LIN {X 0,Y 369.061,Z 354.137,A -85,B 0,C 180,E1 -12856.791,E2 -12856.791} C_VEL
LIN {X 0,Y 369.066,Z 354.138,A -85,B 0,C 180,E1 -12860.132,E2 -12860.132} C_VEL
LIN {X 0,Y 369.162,Z 354.122,A -85,B 0,C 180,E1 -12863.442,E2 -12863.442} C_VEL
LIN {X 0,Y 369.306,Z 354.106,A -85,B 0,C 180,E1 -12867.819,E2 -12867.819} C_VEL
LIN {X 0,Y 369.304,Z 354.11,A -85,B 0,C 180,E1 -12872.182,E2 -12872.182} C_VEL
LIN {X 0,Y 369.16,Z 354.127,A -85,B 0,C 180,E1 -12876.56,E2 -12876.56} C_VEL
LIN {X 0,Y 369.069,Z 354.154,A -85,B 0,C 180,E1 -12879.207,E2 -12879.207} C_VEL
LIN {X 0,Y 370.205,Z 357.177,A -85,B 0,C 180,E1 -12879.375,E2 -12879.375} C_VEL
LIN {X 0,Y 381.684,Z 380.076,A -85,B 0,C 180,E1 -12880.832,E2 -12880.832} C_VEL
LIN {X 0,Y 385.674,Z 389.818,A -85,B 0,C 180,E1 -12881.355,E2 -12881.355} C_VEL
LIN {X 0,Y 382.326,Z 514.998,A -85,B 0,C 180,E1 -12883.86,E2 -12883.86} C_VEL
LIN {X 0,Y 381.61,Z 530.295,A -85,B 0,C 180,E1 -12884.372,E2 -12884.372} C_VEL
LIN {X 0,Y 380.673,Z 545.172,A -85,B 0,C 180,E1 -12885.085,E2 -12885.085} C_VEL
LIN {X 0,Y 379.475,Z 558.92,A -85,B 0,C 180,E1 -12885.948,E2 -12885.948} C_VEL
LIN {X 0,Y 378.337,Z 564.266,A -85,B 0,C 180,E1 -12886.294,E2 -12886.294} C_VEL
LIN {X 0,Y 374.743,Z 572.831,A -85,B 0,C 180,E1 -12886.834,E2 -12886.834} C_VEL
LIN {X 0,Y 371.121,Z 581.153,A -85,B 0,C 180,E1 -12887.454,E2 -12887.454} C_VEL
LIN {X 0,Y 369.922,Z 585.999,A -85,B 0,C 180,E1 -12887.926,E2 -12887.926} C_VEL
LIN {X 0,Y 368.194,Z 599.192,A -85,B 0,C 180,E1 -12889.514,E2 -12889.514} C_VEL
LIN {X 0,Y 366.673,Z 609.996,A -85,B 0,C 180,E1 -12891.092,E2 -12891.092} C_VEL
LIN {X 0,Y 365.196,Z 620.539,A -85,B 0,C 180,E1 -12892.936,E2 -12892.936} C_VEL
LIN {X 0,Y 363.939,Z 629.47,A -85,B 0,C 180,E1 -12894.821,E2 -12894.821} C_VEL
LIN {X 0,Y 362.732,Z 637.87,A -85,B 0,C 180,E1 -12896.967,E2 -12896.967} C_VEL
LIN {X 0,Y 361.879,Z 644.548,A -85,B 0,C 180,E1 -12899.079,E2 -12899.079} C_VEL
LIN {X 0,Y 361.278,Z 649.748,A -85,B 0,C 180,E1 -12901.135,E2 -12901.135} C_VEL
LIN {X 0,Y 360.891,Z 653.719,A -85,B 0,C 180,E1 -12903.134,E2 -12903.134} C_VEL
LIN {X 0,Y 360.521,Z 656.543,A -85,B 0,C 180,E1 -12905.039,E2 -12905.039} C_VEL
LIN {X 0,Y 360.316,Z 658.689,A -85,B 0,C 180,E1 -12907.205,E2 -12907.205} C_VEL
LIN {X 0,Y 360.265,Z 659.556,A -85,B 0,C 180,E1 -12908.71,E2 -12908.71} C_VEL
LIN {X 0,Y 360.246,Z 659.917,A -85,B 0,C 180,E1 -12910.46,E2 -12910.46} C_VEL
LIN {X 0,Y 360.31,Z 659.558,A -85,B 0,C 180,E1 -12912.165,E2 -12912.165} C_VEL
LIN {X 0,Y 360.551,Z 657.956,A -85,B 0,C 180,E1 -12914.566,E2 -12914.566} C_VEL
LIN {X 0,Y 361.005,Z 654.876,A -85,B 0,C 180,E1 -12917.048,E2 -12917.048} C_VEL
LIN {X 0,Y 361.53,Z 650.776,A -85,B 0,C 180,E1 -12919.302,E2 -12919.302} C_VEL
LIN {X 0,Y 362.352,Z 645.097,A -85,B 0,C 180,E1 -12921.635,E2 -12921.635} C_VEL
LIN {X 0,Y 363.361,Z 638.585,A -85,B 0,C 180,E1 -12923.741,E2 -12923.741} C_VEL
LIN {X 0,Y 364.596,Z 631.247,A -85,B 0,C 180,E1 -12925.679,E2 -12925.679} C_VEL
LIN {X 0,Y 366.096,Z 622.256,A -85,B 0,C 180,E1 -12927.638,E2 -12927.638} C_VEL
LIN {X 0,Y 367.793,Z 612.196,A -85,B 0,C 180,E1 -12929.452,E2 -12929.452} C_VEL
LIN {X 0,Y 369.643,Z 600.703,A -85,B 0,C 180,E1 -12931.17,E2 -12931.17} C_VEL
LIN {X 0,Y 371.322,Z 589.315,A -85,B 0,C 180,E1 -12932.586,E2 -12932.586} C_VEL
LIN {X 0,Y 373.074,Z 576.772,A -85,B 0,C 180,E1 -12933.874,E2 -12933.874} C_VEL
LIN {X 0,Y 374.714,Z 562.889,A -85,B 0,C 180,E1 -12935.038,E2 -12935.038} C_VEL
LIN {X 0,Y 376.037,Z 549.259,A -85,B 0,C 180,E1 -12935.946,E2 -12935.946} C_VEL
LIN {X 0,Y 377.167,Z 534.242,A -85,B 0,C 180,E1 -12936.716,E2 -12936.716} C_VEL
LIN {X 0,Y 378.025,Z 519.128,A -85,B 0,C 180,E1 -12937.262,E2 -12937.262} C_VEL
LIN {X 0,Y 379.027,Z 486.351,A -85,B 0,C 180,E1 -12937.99,E2 -12937.99} C_VEL
LIN {X 0,Y 382.012,Z 393.164,A -85,B 0,C 180,E1 -12939.942,E2 -12939.942} C_VEL
LIN {X 0,Y 374.44,Z 377.297,A -85,B 0,C 180,E1 -12941.119,E2 -12941.119} C_VEL
LIN {X 0,Y 367.639,Z 365.381,A -85,B 0,C 180,E1 -12942.189,E2 -12942.189} C_VEL
LIN {X 0,Y 363.906,Z 359.129,A -85,B 0,C 180,E1 -12942.798,E2 -12942.798} C_VEL
LIN {X 0,Y 362.223,Z 356.441,A -85,B 0,C 180,E1 -12943.08,E2 -12943.08} C_VEL
LIN {X 0,Y 361.891,Z 355.027,A -85,B 0,C 180,E1 -12943.209,E2 -12943.209} C_VEL
LIN {X 0,Y 362.003,Z 355.019,A -85,B 0,C 180,E1 -12946.528,E2 -12946.528} C_VEL
LIN {X 0,Y 362.002,Z 355.019,A -85,B 0,C 180,E1 -12949.937,E2 -12949.937} C_VEL
LIN {X 0,Y 362.122,Z 355.001,A -85,B 0,C 180,E1 -12953.312,E2 -12953.312} C_VEL
LIN {X 0,Y 362.268,Z 354.984,A -85,B 0,C 180,E1 -12957.776,E2 -12957.776} C_VEL
LIN {X 0,Y 362.383,Z 354.969,A -85,B 0,C 180,E1 -12960,E2 -12960} C_VEL
LIN {X 0,Y 362.28,Z 354.98,A -85,B 0,C 180,E1 -12962.223,E2 -12962.223} C_VEL
LIN {X 0,Y 362.126,Z 355.001,A -85,B 0,C 180,E1 -12966.687,E2 -12966.687} C_VEL
LIN {X 0,Y 362.003,Z 355.012,A -85,B 0,C 180,E1 -12970.062,E2 -12970.062} C_VEL
LIN {X 0,Y 362,Z 355.017,A -85,B 0,C 180,E1 -12973.898,E2 -12973.898} C_VEL
LIN {X 0,Y 361.93,Z 355.024,A -85,B 0,C 180,E1 -12976.934,E2 -12976.934} C_VEL
LIN {X 0,Y 361.896,Z 355.03,A -85,B 0,C 180,E1 -12980.46,E2 -12980.46} C_VEL
LIN {X 0,Y 361.897,Z 355.025,A -85,B 0,C 180,E1 -12984.113,E2 -12984.113} C_VEL
LIN {X 0,Y 361.945,Z 355.023,A -85,B 0,C 180,E1 -12986.721,E2 -12986.721} C_VEL
LIN {X 0,Y 361.876,Z 355.03,A -85,B 0,C 180,E1 -12990.327,E2 -12990.327} C_VEL
LIN {X 0,Y 361.856,Z 355.036,A -85,B 0,C 180,E1 -12994.28,E2 -12994.28} C_VEL
LIN {X 0,Y 361.865,Z 355.035,A -85,B 0,C 180,E1 -12997.222,E2 -12997.222} C_VEL
LIN {X 0,Y 361.837,Z 355.04,A -85,B 0,C 180,E1 -13000.755,E2 -13000.755} C_VEL
LIN {X 0,Y 361.822,Z 355.041,A -85,B 0,C 180,E1 -13004.367,E2 -13004.367} C_VEL
LIN {X 0,Y 361.838,Z 355.039,A -85,B 0,C 180,E1 -13007.567,E2 -13007.567} C_VEL
LIN {X 0,Y 361.871,Z 355.094,A -85,B 0,C 180,E1 -13010.388,E2 -13010.388} C_VEL
LIN {X 0,Y 365.331,Z 366.466,A -85,B 0,C 180,E1 -13013.39,E2 -13013.39} C_VEL
LIN {X 0,Y 368.142,Z 376.652,A -85,B 0,C 180,E1 -13015.863,E2 -13015.863} C_VEL
LIN {X 0,Y 370.196,Z 385.294,A -85,B 0,C 180,E1 -13017.818,E2 -13017.818} C_VEL
LIN {X 0,Y 374.385,Z 395.128,A -85,B 0,C 180,E1 -13018.521,E2 -13018.521} C_VEL
LIN {X 0,Y 378.827,Z 419.388,A -85,B 0,C 180,E1 -13019.578,E2 -13019.578} C_VEL
LIN {X 0,Y 381.127,Z 434.485,A -85,B 0,C 180,E1 -13020.167,E2 -13020.167} C_VEL
LIN {X 0,Y 377.305,Z 553.846,A -85,B 0,C 180,E1 -13022.66,E2 -13022.66} C_VEL
LIN {X 0,Y 376.29,Z 569.415,A -85,B 0,C 180,E1 -13023.181,E2 -13023.181} C_VEL
LIN {X 0,Y 374.756,Z 585.071,A -85,B 0,C 180,E1 -13023.925,E2 -13023.925} C_VEL
LIN {X 0,Y 373.122,Z 599.399,A -85,B 0,C 180,E1 -13024.834,E2 -13024.834} C_VEL
LIN {X 0,Y 371.252,Z 613.643,A -85,B 0,C 180,E1 -13025.983,E2 -13025.983} C_VEL
LIN {X 0,Y 369.261,Z 627.13,A -85,B 0,C 180,E1 -13027.33,E2 -13027.33} C_VEL
LIN {X 0,Y 367.379,Z 639.47,A -85,B 0,C 180,E1 -13028.833,E2 -13028.833} C_VEL
LIN {X 0,Y 365.686,Z 650.7,A -85,B 0,C 180,E1 -13030.474,E2 -13030.474} C_VEL
LIN {X 0,Y 364.14,Z 661.138,A -85,B 0,C 180,E1 -13032.303,E2 -13032.303} C_VEL
LIN {X 0,Y 362.777,Z 670.461,A -85,B 0,C 180,E1 -13034.263,E2 -13034.263} C_VEL
LIN {X 0,Y 361.798,Z 678.215,A -85,B 0,C 180,E1 -13036.23,E2 -13036.23} C_VEL
LIN {X 0,Y 361.144,Z 684.684,A -85,B 0,C 180,E1 -13038.209,E2 -13038.209} C_VEL
LIN {X 0,Y 360.631,Z 690.639,A -85,B 0,C 180,E1 -13040.465,E2 -13040.465} C_VEL
LIN {X 0,Y 360.485,Z 694.219,A -85,B 0,C 180,E1 -13042.156,E2 -13042.156} C_VEL
LIN {X 0,Y 360.396,Z 697.799,A -85,B 0,C 180,E1 -13044.404,E2 -13044.404} C_VEL
LIN {X 0,Y 360.38,Z 700.136,A -85,B 0,C 180,E1 -13046.646,E2 -13046.646} C_VEL
LIN {X 0,Y 360.529,Z 701.285,A -85,B 0,C 180,E1 -13048.883,E2 -13048.883} C_VEL
LIN {X 0,Y 360.529,Z 701.244,A -85,B 0,C 180,E1 -13051.116,E2 -13051.116} C_VEL
LIN {X 0,Y 360.387,Z 699.974,A -85,B 0,C 180,E1 -13053.353,E2 -13053.353} C_VEL
LIN {X 0,Y 360.386,Z 697.46,A -85,B 0,C 180,E1 -13055.595,E2 -13055.595} C_VEL
LIN {X 0,Y 360.479,Z 693.683,A -85,B 0,C 180,E1 -13057.843,E2 -13057.843} C_VEL
LIN {X 0,Y 360.693,Z 688.544,A -85,B 0,C 180,E1 -13060.099,E2 -13060.099} C_VEL
LIN {X 0,Y 361.292,Z 681.924,A -85,B 0,C 180,E1 -13062.355,E2 -13062.355} C_VEL
LIN {X 0,Y 362.189,Z 673.631,A -85,B 0,C 180,E1 -13064.61,E2 -13064.61} C_VEL
LIN {X 0,Y 363.223,Z 664.766,A -85,B 0,C 180,E1 -13066.582,E2 -13066.582} C_VEL
LIN {X 0,Y 364.739,Z 654.106,A -85,B 0,C 180,E1 -13068.537,E2 -13068.537} C_VEL
LIN {X 0,Y 366.115,Z 643.14,A -85,B 0,C 180,E1 -13070.214,E2 -13070.214} C_VEL
LIN {X 0,Y 367.699,Z 631.184,A -85,B 0,C 180,E1 -13071.735,E2 -13071.735} C_VEL
LIN {X 0,Y 369.248,Z 619.571,A -85,B 0,C 180,E1 -13072.965,E2 -13072.965} C_VEL
LIN {X 0,Y 371.086,Z 605.528,A -85,B 0,C 180,E1 -13074.176,E2 -13074.176} C_VEL
LIN {X 0,Y 372.586,Z 591.611,A -85,B 0,C 180,E1 -13075.138,E2 -13075.138} C_VEL
LIN {X 0,Y 373.905,Z 577.102,A -85,B 0,C 180,E1 -13075.913,E2 -13075.913} C_VEL
LIN {X 0,Y 374.933,Z 562.841,A -85,B 0,C 180,E1 -13076.472,E2 -13076.472} C_VEL
LIN {X 0,Y 375.62,Z 547.531,A -85,B 0,C 180,E1 -13076.87,E2 -13076.87} C_VEL
LIN {X 0,Y 378.618,Z 434.526,A -85,B 0,C 180,E1 -13079.154,E2 -13079.154} C_VEL
LIN {X 0,Y 373.667,Z 404.594,A -85,B 0,C 180,E1 -13080.216,E2 -13080.216} C_VEL
LIN {X 0,Y 370.766,Z 389.788,A -85,B 0,C 180,E1 -13080.796,E2 -13080.796} C_VEL
LIN {X 0,Y 370.286,Z 388.239,A -85,B 0,C 180,E1 -13080.906,E2 -13080.906} C_VEL
LIN {X 0,Y 367.141,Z 374.609,A -85,B 0,C 180,E1 -13083.719,E2 -13083.719} C_VEL
LIN {X 0,Y 362.919,Z 358.954,A -85,B 0,C 180,E1 -13087.167,E2 -13087.167} C_VEL
LIN {X 0,Y 361.884,Z 355.037,A -85,B 0,C 180,E1 -13088.077,E2 -13088.077} C_VEL
LIN {X 0,Y 361.825,Z 355.042,A -85,B 0,C 180,E1 -13091.33,E2 -13091.33} C_VEL
LIN {X 0,Y 361.832,Z 355.035,A -85,B 0,C 180,E1 -13094.365,E2 -13094.365} C_VEL
LIN {X 0,Y 361.833,Z 355.037,A -85,B 0,C 180,E1 -13097.568,E2 -13097.568} C_VEL
LIN {X 0,Y 361.867,Z 355.035,A -85,B 0,C 180,E1 -13100.973,E2 -13100.973} C_VEL
LIN {X 0,Y 361.871,Z 355.032,A -85,B 0,C 180,E1 -13104.655,E2 -13104.655} C_VEL
LIN {X 0,Y 361.834,Z 355.035,A -85,B 0,C 180,E1 -13108.371,E2 -13108.371} C_VEL
LIN {X 0,Y 361.897,Z 355.032,A -85,B 0,C 180,E1 -13110.955,E2 -13110.955} C_VEL
LIN {X 0,Y 361.951,Z 355.023,A -85,B 0,C 180,E1 -13113.475,E2 -13113.475} C_VEL
LIN {X 0,Y 361.887,Z 355.034,A -85,B 0,C 180,E1 -13117.145,E2 -13117.145} C_VEL
LIN {X 0,Y 361.903,Z 355.029,A -85,B 0,C 180,E1 -13120.724,E2 -13120.724} C_VEL
LIN {X 0,Y 361.93,Z 355.029,A -85,B 0,C 180,E1 -13123.066,E2 -13123.066} C_VEL
LIN {X 0,Y 361.995,Z 355.016,A -85,B 0,C 180,E1 -13126.528,E2 -13126.528} C_VEL
LIN {X 0,Y 362.028,Z 355.01,A -85,B 0,C 180,E1 -13129.938,E2 -13129.938} C_VEL
LIN {X 0,Y 362.158,Z 354.997,A -85,B 0,C 180,E1 -13133.314,E2 -13133.314} C_VEL
LIN {X 0,Y 362.28,Z 354.979,A -85,B 0,C 180,E1 -13137.777,E2 -13137.777} C_VEL
LIN {X 0,Y 362.425,Z 354.961,A -85,B 0,C 180,E1 -13140,E2 -13140} C_VEL
LIN {X 0,Y 362.28,Z 354.98,A -85,B 0,C 180,E1 -13142.224,E2 -13142.224} C_VEL
LIN {X 0,Y 362.17,Z 354.997,A -85,B 0,C 180,E1 -13146.687,E2 -13146.687} C_VEL
LIN {X 0,Y 362.072,Z 355.011,A -85,B 0,C 180,E1 -13148.934,E2 -13148.934} C_VEL
LIN {X 0,Y 361.958,Z 355.021,A -85,B 0,C 180,E1 -13152.333,E2 -13152.333} C_VEL
LIN {X 0,Y 361.96,Z 355.023,A -85,B 0,C 180,E1 -13154.621,E2 -13154.621} C_VEL
LIN {X 0,Y 361.958,Z 355.02,A -85,B 0,C 180,E1 -13158.1,E2 -13158.1} C_VEL
LIN {X 0,Y 361.859,Z 355.032,A -85,B 0,C 180,E1 -13161.655,E2 -13161.655} C_VEL
LIN {X 0,Y 361.924,Z 355.024,A -85,B 0,C 180,E1 -13165.291,E2 -13165.291} C_VEL
LIN {X 0,Y 361.917,Z 355.024,A -85,B 0,C 180,E1 -13167.779,E2 -13167.779} C_VEL
LIN {X 0,Y 361.845,Z 355.034,A -85,B 0,C 180,E1 -13171.286,E2 -13171.286} C_VEL
LIN {X 0,Y 361.853,Z 355.035,A -85,B 0,C 180,E1 -13174.281,E2 -13174.281} C_VEL
LIN {X 0,Y 361.862,Z 355.032,A -85,B 0,C 180,E1 -13177.223,E2 -13177.223} C_VEL
LIN {X 0,Y 361.833,Z 355.04,A -85,B 0,C 180,E1 -13180.756,E2 -13180.756} C_VEL
LIN {X 0,Y 361.816,Z 355.041,A -85,B 0,C 180,E1 -13184.369,E2 -13184.369} C_VEL
LIN {X 0,Y 361.832,Z 355.035,A -85,B 0,C 180,E1 -13187.57,E2 -13187.57} C_VEL
LIN {X 0,Y 361.864,Z 355.033,A -85,B 0,C 180,E1 -13190.975,E2 -13190.975} C_VEL
LIN {X 0,Y 361.875,Z 355.035,A -85,B 0,C 180,E1 -13194.656,E2 -13194.656} C_VEL
LIN {X 0,Y 361.839,Z 355.039,A -85,B 0,C 180,E1 -13198.371,E2 -13198.371} C_VEL
LIN {X 0,Y 361.867,Z 355.032,A -85,B 0,C 180,E1 -13200.953,E2 -13200.953} C_VEL
LIN {X 0,Y 361.897,Z 355.03,A -85,B 0,C 180,E1 -13204.708,E2 -13204.708} C_VEL
LIN {X 0,Y 361.894,Z 355.033,A -85,B 0,C 180,E1 -13208.348,E2 -13208.348} C_VEL
LIN {X 0,Y 361.907,Z 355.029,A -85,B 0,C 180,E1 -13212.093,E2 -13212.093} C_VEL
LIN {X 0,Y 361.983,Z 355.02,A -85,B 0,C 180,E1 -13216.114,E2 -13216.114} C_VEL
LIN {X 0,Y 362.003,Z 355.016,A -85,B 0,C 180,E1 -13219.938,E2 -13219.938} C_VEL
LIN {X 0,Y 362.125,Z 354.998,A -85,B 0,C 180,E1 -13223.313,E2 -13223.313} C_VEL
LIN {X 0,Y 362.268,Z 354.982,A -85,B 0,C 180,E1 -13227.777,E2 -13227.777} C_VEL
LIN {X 0,Y 362.195,Z 354.99,A -85,B 0,C 180,E1 -13231.112,E2 -13231.112} C_VEL
LIN {X 0,Y 362.267,Z 354.987,A -85,B 0,C 180,E1 -13232.224,E2 -13232.224} C_VEL
LIN {X 0,Y 362.125,Z 355.003,A -85,B 0,C 180,E1 -13236.688,E2 -13236.688} C_VEL
LIN {X 0,Y 362.068,Z 355.008,A -85,B 0,C 180,E1 -13238.599,E2 -13238.599} C_VEL
LIN {X 0,Y 363.202,Z 358.066,A -85,B 0,C 180,E1 -13238.792,E2 -13238.792} C_VEL
LIN {X 0,Y 375.716,Z 382.87,A -85,B 0,C 180,E1 -13240.426,E2 -13240.426} C_VEL
LIN {X 0,Y 379.276,Z 391.483,A -85,B 0,C 180,E1 -13240.904,E2 -13240.904} C_VEL
LIN {X 0,Y 375.837,Z 515.861,A -85,B 0,C 180,E1 -13243.443,E2 -13243.443} C_VEL
LIN {X 0,Y 375.108,Z 530.746,A -85,B 0,C 180,E1 -13243.951,E2 -13243.951} C_VEL
LIN {X 0,Y 374.11,Z 545.881,A -85,B 0,C 180,E1 -13244.692,E2 -13244.692} C_VEL
LIN {X 0,Y 372.819,Z 560.212,A -85,B 0,C 180,E1 -13245.612,E2 -13245.612} C_VEL
LIN {X 0,Y 371.331,Z 574.464,A -85,B 0,C 180,E1 -13246.776,E2 -13246.776} C_VEL
LIN {X 0,Y 369.922,Z 585.999,A -85,B 0,C 180,E1 -13247.926,E2 -13247.926} C_VEL
LIN {X 0,Y 368.73,Z 590.809,A -85,B 0,C 180,E1 -13248.424,E2 -13248.424} C_VEL
LIN {X 0,Y 365.027,Z 598.445,A -85,B 0,C 180,E1 -13249.224,E2 -13249.224} C_VEL
LIN {X 0,Y 361.249,Z 605.781,A -85,B 0,C 180,E1 -13250.096,E2 -13250.096} C_VEL
LIN {X 0,Y 359.922,Z 610.01,A -85,B 0,C 180,E1 -13250.717,E2 -13250.717} C_VEL
LIN {X 0,Y 358.5,Z 619.679,A -85,B 0,C 180,E1 -13252.416,E2 -13252.416} C_VEL
LIN {X 0,Y 357.085,Z 629.183,A -85,B 0,C 180,E1 -13254.414,E2 -13254.414} C_VEL
LIN {X 0,Y 355.95,Z 636.912,A -85,B 0,C 180,E1 -13256.376,E2 -13256.376} C_VEL
LIN {X 0,Y 355.098,Z 643.383,A -85,B 0,C 180,E1 -13258.36,E2 -13258.36} C_VEL
LIN {X 0,Y 354.428,Z 648.754,A -85,B 0,C 180,E1 -13260.375,E2 -13260.375} C_VEL
LIN {X 0,Y 353.956,Z 653.014,A -85,B 0,C 180,E1 -13262.419,E2 -13262.419} C_VEL
LIN {X 0,Y 353.653,Z 655.352,A -85,B 0,C 180,E1 -13263.81,E2 -13263.81} C_VEL
LIN {X 0,Y 353.383,Z 657.437,A -85,B 0,C 180,E1 -13265.372,E2 -13265.372} C_VEL
LIN {X 0,Y 353.236,Z 659.153,A -85,B 0,C 180,E1 -13267.264,E2 -13267.264} C_VEL
LIN {X 0,Y 353.174,Z 660.209,A -85,B 0,C 180,E1 -13269.553,E2 -13269.553} C_VEL
LIN {X 0,Y 353.164,Z 660.276,A -85,B 0,C 180,E1 -13271.049,E2 -13271.049} C_VEL
LIN {X 0,Y 353.277,Z 659.841,A -85,B 0,C 180,E1 -13272.602,E2 -13272.602} C_VEL
LIN {X 0,Y 353.438,Z 658.764,A -85,B 0,C 180,E1 -13274.287,E2 -13274.287} C_VEL
LIN {X 0,Y 353.712,Z 657.053,A -85,B 0,C 180,E1 -13275.938,E2 -13275.938} C_VEL
LIN {X 0,Y 354.205,Z 653.593,A -85,B 0,C 180,E1 -13278.277,E2 -13278.277} C_VEL
LIN {X 0,Y 354.933,Z 648.636,A -85,B 0,C 180,E1 -13280.681,E2 -13280.681} C_VEL
LIN {X 0,Y 355.931,Z 642.421,A -85,B 0,C 180,E1 -13282.984,E2 -13282.984} C_VEL
LIN {X 0,Y 357.252,Z 634.831,A -85,B 0,C 180,E1 -13285.214,E2 -13285.214} C_VEL
LIN {X 0,Y 358.826,Z 625.761,A -85,B 0,C 180,E1 -13287.374,E2 -13287.374} C_VEL
LIN {X 0,Y 360.668,Z 615.655,A -85,B 0,C 180,E1 -13289.338,E2 -13289.338} C_VEL
LIN {X 0,Y 362.593,Z 604.2,A -85,B 0,C 180,E1 -13291.174,E2 -13291.174} C_VEL
LIN {X 0,Y 364.398,Z 592.713,A -85,B 0,C 180,E1 -13292.698,E2 -13292.698} C_VEL
LIN {X 0,Y 366.316,Z 579.85,A -85,B 0,C 180,E1 -13294.102,E2 -13294.102} C_VEL
LIN {X 0,Y 368.057,Z 566.624,A -85,B 0,C 180,E1 -13295.278,E2 -13295.278} C_VEL
LIN {X 0,Y 369.388,Z 554.086,A -85,B 0,C 180,E1 -13296.193,E2 -13296.193} C_VEL
LIN {X 0,Y 370.715,Z 538.8,A -85,B 0,C 180,E1 -13297.056,E2 -13297.056} C_VEL
LIN {X 0,Y 371.681,Z 523.341,A -85,B 0,C 180,E1 -13297.687,E2 -13297.687} C_VEL
LIN {X 0,Y 372.417,Z 505.938,A -85,B 0,C 180,E1 -13298.135,E2 -13298.135} C_VEL
LIN {X 0,Y 376.125,Z 395.564,A -85,B 0,C 180,E1 -13300.477,E2 -13300.477} C_VEL
LIN {X 0,Y 368.653,Z 379.876,A -85,B 0,C 180,E1 -13301.689,E2 -13301.689} C_VEL
LIN {X 0,Y 361.434,Z 367.372,A -85,B 0,C 180,E1 -13302.874,E2 -13302.874} C_VEL
LIN {X 0,Y 356.643,Z 359.777,A -85,B 0,C 180,E1 -13303.691,E2 -13303.691} C_VEL
LIN {X 0,Y 355.166,Z 357.264,A -85,B 0,C 180,E1 -13303.953,E2 -13303.953} C_VEL
LIN {X 0,Y 354.87,Z 355.91,A -85,B 0,C 180,E1 -13304.05,E2 -13304.05} C_VEL
LIN {X 0,Y 354.924,Z 355.9,A -85,B 0,C 180,E1 -13307.419,E2 -13307.419} C_VEL
LIN {X 0,Y 354.997,Z 355.889,A -85,B 0,C 180,E1 -13310.887,E2 -13310.887} C_VEL
LIN {X 0,Y 355.065,Z 355.881,A -85,B 0,C 180,E1 -13314.32,E2 -13314.32} C_VEL
LIN {X 0,Y 355.23,Z 355.861,A -85,B 0,C 180,E1 -13317.732,E2 -13317.732} C_VEL
LIN {X 0,Y 355.334,Z 355.847,A -85,B 0,C 180,E1 -13320,E2 -13320} C_VEL
LIN {X 0,Y 355.243,Z 355.856,A -85,B 0,C 180,E1 -13322.267,E2 -13322.267} C_VEL
LIN {X 0,Y 355.092,Z 355.876,A -85,B 0,C 180,E1 -13326.82,E2 -13326.82} C_VEL
LIN {X 0,Y 354.959,Z 355.889,A -85,B 0,C 180,E1 -13330.264,E2 -13330.264} C_VEL
LIN {X 0,Y 354.945,Z 355.896,A -85,B 0,C 180,E1 -13334.018,E2 -13334.018} C_VEL
LIN {X 0,Y 354.892,Z 355.898,A -85,B 0,C 180,E1 -13338.092,E2 -13338.092} C_VEL
LIN {X 0,Y 354.837,Z 355.907,A -85,B 0,C 180,E1 -13342.106,E2 -13342.106} C_VEL
LIN {X 0,Y 354.902,Z 355.902,A -85,B 0,C 180,E1 -13345.827,E2 -13345.827} C_VEL
LIN {X 0,Y 354.856,Z 355.903,A -85,B 0,C 180,E1 -13349.678,E2 -13349.678} C_VEL
LIN {X 0,Y 354.808,Z 355.915,A -85,B 0,C 180,E1 -13353.701,E2 -13353.701} C_VEL
LIN {X 0,Y 354.799,Z 355.917,A -85,B 0,C 180,E1 -13356.459,E2 -13356.459} C_VEL
LIN {X 0,Y 354.825,Z 355.912,A -85,B 0,C 180,E1 -13359.423,E2 -13359.423} C_VEL
LIN {X 0,Y 354.789,Z 355.916,A -85,B 0,C 180,E1 -13362.867,E2 -13362.867} C_VEL
LIN {X 0,Y 354.783,Z 355.917,A -85,B 0,C 180,E1 -13366.105,E2 -13366.105} C_VEL
LIN {X 0,Y 354.827,Z 356.042,A -85,B 0,C 180,E1 -13369.601,E2 -13369.601} C_VEL
LIN {X 0,Y 358.395,Z 367.431,A -85,B 0,C 180,E1 -13372.747,E2 -13372.747} C_VEL
LIN {X 0,Y 361.114,Z 377.388,A -85,B 0,C 180,E1 -13375.248,E2 -13375.248} C_VEL
LIN {X 0,Y 362.953,Z 384.928,A -85,B 0,C 180,E1 -13376.978,E2 -13376.978} C_VEL
LIN {X 0,Y 368.684,Z 397.433,A -85,B 0,C 180,E1 -13377.966,E2 -13377.966} C_VEL
LIN {X 0,Y 372.632,Z 419.027,A -85,B 0,C 180,E1 -13378.943,E2 -13378.943} C_VEL
LIN {X 0,Y 375.098,Z 435.7,A -85,B 0,C 180,E1 -13379.61,E2 -13379.61} C_VEL
LIN {X 0,Y 371.193,Z 552.556,A -85,B 0,C 180,E1 -13382.094,E2 -13382.094} C_VEL
LIN {X 0,Y 370.111,Z 568.367,A -85,B 0,C 180,E1 -13382.62,E2 -13382.62} C_VEL
LIN {X 0,Y 368.516,Z 584.175,A -85,B 0,C 180,E1 -13383.373,E2 -13383.373} C_VEL
LIN {X 0,Y 366.857,Z 598.388,A -85,B 0,C 180,E1 -13384.28,E2 -13384.28} C_VEL
LIN {X 0,Y 364.956,Z 612.161,A -85,B 0,C 180,E1 -13385.39,E2 -13385.39} C_VEL
LIN {X 0,Y 362.891,Z 625.845,A -85,B 0,C 180,E1 -13386.759,E2 -13386.759} C_VEL
LIN {X 0,Y 360.868,Z 638.321,A -85,B 0,C 180,E1 -13388.282,E2 -13388.282} C_VEL
LIN {X 0,Y 359.108,Z 649.603,A -85,B 0,C 180,E1 -13389.949,E2 -13389.949} C_VEL
LIN {X 0,Y 357.336,Z 660.88,A -85,B 0,C 180,E1 -13391.954,E2 -13391.954} C_VEL
LIN {X 0,Y 355.852,Z 670.176,A -85,B 0,C 180,E1 -13393.948,E2 -13393.948} C_VEL
LIN {X 0,Y 354.673,Z 678.947,A -85,B 0,C 180,E1 -13396.244,E2 -13396.244} C_VEL
LIN {X 0,Y 353.96,Z 686.021,A -85,B 0,C 180,E1 -13398.547,E2 -13398.547} C_VEL
LIN {X 0,Y 353.513,Z 691.598,A -85,B 0,C 180,E1 -13400.848,E2 -13400.848} C_VEL
LIN {X 0,Y 353.367,Z 695.803,A -85,B 0,C 180,E1 -13403.146,E2 -13403.146} C_VEL
LIN {X 0,Y 353.302,Z 698.735,A -85,B 0,C 180,E1 -13405.436,E2 -13405.436} C_VEL
LIN {X 0,Y 353.387,Z 700.459,A -85,B 0,C 180,E1 -13407.72,E2 -13407.72} C_VEL
LIN {X 0,Y 353.452,Z 700.997,A -85,B 0,C 180,E1 -13409.999,E2 -13409.999} C_VEL
LIN {X 0,Y 353.405,Z 700.339,A -85,B 0,C 180,E1 -13412.279,E2 -13412.279} C_VEL
LIN {X 0,Y 353.318,Z 698.427,A -85,B 0,C 180,E1 -13414.563,E2 -13414.563} C_VEL
LIN {X 0,Y 353.379,Z 695.269,A -85,B 0,C 180,E1 -13416.853,E2 -13416.853} C_VEL
LIN {X 0,Y 353.507,Z 690.797,A -85,B 0,C 180,E1 -13419.151,E2 -13419.151} C_VEL
LIN {X 0,Y 353.956,Z 684.908,A -85,B 0,C 180,E1 -13421.452,E2 -13421.452} C_VEL
LIN {X 0,Y 354.671,Z 677.441,A -85,B 0,C 180,E1 -13423.755,E2 -13423.755} C_VEL
LIN {X 0,Y 355.64,Z 669.431,A -85,B 0,C 180,E1 -13425.766,E2 -13425.766} C_VEL
LIN {X 0,Y 356.977,Z 659.793,A -85,B 0,C 180,E1 -13427.767,E2 -13427.767} C_VEL
LIN {X 0,Y 358.516,Z 648.805,A -85,B 0,C 180,E1 -13429.655,E2 -13429.655} C_VEL
LIN {X 0,Y 360.141,Z 637.179,A -85,B 0,C 180,E1 -13431.312,E2 -13431.312} C_VEL
LIN {X 0,Y 361.653,Z 626.706,A -85,B 0,C 180,E1 -13432.569,E2 -13432.569} C_VEL
LIN {X 0,Y 363.294,Z 614.29,A -85,B 0,C 180,E1 -13433.817,E2 -13433.817} C_VEL
LIN {X 0,Y 364.954,Z 600.874,A -85,B 0,C 180,E1 -13434.913,E2 -13434.913} C_VEL
LIN {X 0,Y 366.531,Z 585.687,A -85,B 0,C 180,E1 -13435.895,E2 -13435.895} C_VEL
LIN {X 0,Y 367.852,Z 570.136,A -85,B 0,C 180,E1 -13436.639,E2 -13436.639} C_VEL
LIN {X 0,Y 368.815,Z 555.08,A -85,B 0,C 180,E1 -13437.138,E2 -13437.138} C_VEL
LIN {X 0,Y 372.252,Z 435.303,A -85,B 0,C 180,E1 -13439.621,E2 -13439.621} C_VEL
LIN {X 0,Y 366.631,Z 401.54,A -85,B 0,C 180,E1 -13440.862,E2 -13440.862} C_VEL
LIN {X 0,Y 364.597,Z 391.763,A -85,B 0,C 180,E1 -13441.267,E2 -13441.267} C_VEL
LIN {X 0,Y 363.026,Z 387.923,A -85,B 0,C 180,E1 -13441.513,E2 -13441.513} C_VEL
LIN {X 0,Y 359.64,Z 373.777,A -85,B 0,C 180,E1 -13444.52,E2 -13444.52} C_VEL
LIN {X 0,Y 355.736,Z 359.334,A -85,B 0,C 180,E1 -13447.792,E2 -13447.792} C_VEL
LIN {X 0,Y 354.835,Z 355.917,A -85,B 0,C 180,E1 -13448.6,E2 -13448.6} C_VEL
LIN {X 0,Y 354.792,Z 355.913,A -85,B 0,C 180,E1 -13452.337,E2 -13452.337} C_VEL
LIN {X 0,Y 354.797,Z 355.915,A -85,B 0,C 180,E1 -13455.487,E2 -13455.487} C_VEL
LIN {X 0,Y 354.785,Z 355.919,A -85,B 0,C 180,E1 -13459.179,E2 -13459.179} C_VEL
LIN {X 0,Y 354.805,Z 355.91,A -85,B 0,C 180,E1 -13462.402,E2 -13462.402} C_VEL
LIN {X 0,Y 354.809,Z 355.915,A -85,B 0,C 180,E1 -13464.941,E2 -13464.941} C_VEL
LIN {X 0,Y 354.789,Z 355.913,A -85,B 0,C 180,E1 -13468.405,E2 -13468.405} C_VEL
LIN {X 0,Y 354.847,Z 355.907,A -85,B 0,C 180,E1 -13471.619,E2 -13471.619} C_VEL
LIN {X 0,Y 354.896,Z 355.899,A -85,B 0,C 180,E1 -13474.173,E2 -13474.173} C_VEL
LIN {X 0,Y 354.831,Z 355.907,A -85,B 0,C 180,E1 -13477.894,E2 -13477.894} C_VEL
LIN {X 0,Y 354.919,Z 355.896,A -85,B 0,C 180,E1 -13481.892,E2 -13481.892} C_VEL
LIN {X 0,Y 354.939,Z 355.893,A -85,B 0,C 180,E1 -13485.981,E2 -13485.981} C_VEL
LIN {X 0,Y 354.975,Z 355.888,A -85,B 0,C 180,E1 -13489.736,E2 -13489.736} C_VEL
LIN {X 0,Y 355.122,Z 355.875,A -85,B 0,C 180,E1 -13493.181,E2 -13493.181} C_VEL
LIN {X 0,Y 355.243,Z 355.855,A -85,B 0,C 180,E1 -13497.733,E2 -13497.733} C_VEL
LIN {X 0,Y 355.395,Z 355.836,A -85,B 0,C 180,E1 -13500,E2 -13500} C_VEL
LIN {X 0,Y 355.243,Z 355.857,A -85,B 0,C 180,E1 -13502.268,E2 -13502.268} C_VEL
LIN {X 0,Y 355.136,Z 355.874,A -85,B 0,C 180,E1 -13506.82,E2 -13506.82} C_VEL
LIN {X 0,Y 355.013,Z 355.888,A -85,B 0,C 180,E1 -13509.113,E2 -13509.113} C_VEL
LIN {X 0,Y 354.919,Z 355.9,A -85,B 0,C 180,E1 -13512.581,E2 -13512.581} C_VEL
LIN {X 0,Y 354.888,Z 355.899,A -85,B 0,C 180,E1 -13516.097,E2 -13516.097} C_VEL
LIN {X 0,Y 354.905,Z 355.9,A -85,B 0,C 180,E1 -13518.472,E2 -13518.472} C_VEL
LIN {X 0,Y 354.814,Z 355.91,A -85,B 0,C 180,E1 -13522.108,E2 -13522.108} C_VEL
LIN {X 0,Y 354.896,Z 355.897,A -85,B 0,C 180,E1 -13525.828,E2 -13525.828} C_VEL
LIN {X 0,Y 354.853,Z 355.904,A -85,B 0,C 180,E1 -13529.679,E2 -13529.679} C_VEL
LIN {X 0,Y 354.805,Z 355.91,A -85,B 0,C 180,E1 -13533.703,E2 -13533.703} C_VEL
LIN {X 0,Y 354.797,Z 355.915,A -85,B 0,C 180,E1 -13536.46,E2 -13536.46} C_VEL
LIN {X 0,Y 354.824,Z 355.908,A -85,B 0,C 180,E1 -13539.424,E2 -13539.424} C_VEL
LIN {X 0,Y 354.787,Z 355.915,A -85,B 0,C 180,E1 -13542.868,E2 -13542.868} C_VEL
LIN {X 0,Y 354.767,Z 355.917,A -85,B 0,C 180,E1 -13546.104,E2 -13546.104} C_VEL
LIN {X 0,Y 354.783,Z 355.914,A -85,B 0,C 180,E1 -13549.179,E2 -13549.179} C_VEL
LIN {X 0,Y 354.806,Z 355.914,A -85,B 0,C 180,E1 -13552.404,E2 -13552.404} C_VEL
LIN {X 0,Y 354.813,Z 355.912,A -85,B 0,C 180,E1 -13554.942,E2 -13554.942} C_VEL
LIN {X 0,Y 354.795,Z 355.917,A -85,B 0,C 180,E1 -13558.406,E2 -13558.406} C_VEL
LIN {X 0,Y 354.804,Z 355.911,A -85,B 0,C 180,E1 -13561.616,E2 -13561.616} C_VEL
LIN {X 0,Y 354.854,Z 355.904,A -85,B 0,C 180,E1 -13565.424,E2 -13565.424} C_VEL
LIN {X 0,Y 354.841,Z 355.906,A -85,B 0,C 180,E1 -13569.115,E2 -13569.115} C_VEL
LIN {X 0,Y 354.854,Z 355.907,A -85,B 0,C 180,E1 -13572.718,E2 -13572.718} C_VEL
LIN {X 0,Y 354.943,Z 355.899,A -85,B 0,C 180,E1 -13576.255,E2 -13576.255} C_VEL
LIN {X 0,Y 354.959,Z 355.892,A -85,B 0,C 180,E1 -13579.736,E2 -13579.736} C_VEL
LIN {X 0,Y 355.091,Z 355.875,A -85,B 0,C 180,E1 -13583.18,E2 -13583.18} C_VEL
LIN {X 0,Y 355.231,Z 355.859,A -85,B 0,C 180,E1 -13587.733,E2 -13587.733} C_VEL
LIN {X 0,Y 355.165,Z 355.866,A -85,B 0,C 180,E1 -13591.134,E2 -13591.134} C_VEL
LIN {X 0,Y 355.229,Z 355.863,A -85,B 0,C 180,E1 -13592.268,E2 -13592.268} C_VEL
LIN {X 0,Y 355.092,Z 355.879,A -85,B 0,C 180,E1 -13596.821,E2 -13596.821} C_VEL
LIN {X 0,Y 355.078,Z 355.882,A -85,B 0,C 180,E1 -13598,E2 -13598} C_VEL
LIN {X 0,Y 356.091,Z 358.713,A -85,B 0,C 180,E1 -13598.174,E2 -13598.174} C_VEL
LIN {X 0,Y 369.134,Z 384.486,A -85,B 0,C 180,E1 -13599.927,E2 -13599.927} C_VEL
LIN {X 0,Y 372.925,Z 393.263,A -85,B 0,C 180,E1 -13600.442,E2 -13600.442} C_VEL
LIN {X 0,Y 369.388,Z 515.929,A -85,B 0,C 180,E1 -13602.988,E2 -13602.988} C_VEL
LIN {X 0,Y 368.628,Z 530.956,A -85,B 0,C 180,E1 -13603.507,E2 -13603.507} C_VEL
LIN {X 0,Y 367.599,Z 546.04,A -85,B 0,C 180,E1 -13604.254,E2 -13604.254} C_VEL
LIN {X 0,Y 366.296,Z 559.951,A -85,B 0,C 180,E1 -13605.155,E2 -13605.155} C_VEL
LIN {X 0,Y 364.937,Z 573.084,A -85,B 0,C 180,E1 -13606.229,E2 -13606.229} C_VEL
LIN {X 0,Y 363.194,Z 586.794,A -85,B 0,C 180,E1 -13607.599,E2 -13607.599} C_VEL
LIN {X 0,Y 361.483,Z 599.444,A -85,B 0,C 180,E1 -13609.154,E2 -13609.154} C_VEL
LIN {X 0,Y 359.922,Z 610.01,A -85,B 0,C 180,E1 -13610.717,E2 -13610.717} C_VEL
LIN {X 0,Y 358.617,Z 614.15,A -85,B 0,C 180,E1 -13611.358,E2 -13611.358} C_VEL
LIN {X 0,Y 354.852,Z 620.634,A -85,B 0,C 180,E1 -13612.404,E2 -13612.404} C_VEL
LIN {X 0,Y 351.207,Z 626.766,A -85,B 0,C 180,E1 -13613.53,E2 -13613.53} C_VEL
LIN {X 0,Y 350.104,Z 630.162,A -85,B 0,C 180,E1 -13614.29,E2 -13614.29} C_VEL
LIN {X 0,Y 348.899,Z 637.849,A -85,B 0,C 180,E1 -13616.306,E2 -13616.306} C_VEL
LIN {X 0,Y 348.019,Z 644.223,A -85,B 0,C 180,E1 -13618.332,E2 -13618.332} C_VEL
LIN {X 0,Y 347.351,Z 649.513,A -85,B 0,C 180,E1 -13620.387,E2 -13620.387} C_VEL
LIN {X 0,Y 346.87,Z 653.718,A -85,B 0,C 180,E1 -13622.475,E2 -13622.475} C_VEL
LIN {X 0,Y 346.426,Z 656.956,A -85,B 0,C 180,E1 -13624.614,E2 -13624.614} C_VEL
LIN {X 0,Y 346.21,Z 658.582,A -85,B 0,C 180,E1 -13626.065,E2 -13626.065} C_VEL
LIN {X 0,Y 346.121,Z 659.84,A -85,B 0,C 180,E1 -13627.636,E2 -13627.636} C_VEL
LIN {X 0,Y 346.094,Z 660.606,A -85,B 0,C 180,E1 -13629.497,E2 -13629.497} C_VEL
LIN {X 0,Y 346.095,Z 660.675,A -85,B 0,C 180,E1 -13631.292,E2 -13631.292} C_VEL
LIN {X 0,Y 346.277,Z 659.73,A -85,B 0,C 180,E1 -13633.635,E2 -13633.635} C_VEL
LIN {X 0,Y 346.513,Z 658.439,A -85,B 0,C 180,E1 -13635.225,E2 -13635.225} C_VEL
LIN {X 0,Y 346.811,Z 656.569,A -85,B 0,C 180,E1 -13636.847,E2 -13636.847} C_VEL
LIN {X 0,Y 347.347,Z 652.949,A -85,B 0,C 180,E1 -13639.09,E2 -13639.09} C_VEL
LIN {X 0,Y 348.088,Z 648.324,A -85,B 0,C 180,E1 -13641.251,E2 -13641.251} C_VEL
LIN {X 0,Y 349.207,Z 641.875,A -85,B 0,C 180,E1 -13643.613,E2 -13643.613} C_VEL
LIN {X 0,Y 350.644,Z 634.153,A -85,B 0,C 180,E1 -13645.86,E2 -13645.86} C_VEL
LIN {X 0,Y 352.076,Z 626.375,A -85,B 0,C 180,E1 -13647.725,E2 -13647.725} C_VEL
LIN {X 0,Y 353.856,Z 617.113,A -85,B 0,C 180,E1 -13649.579,E2 -13649.579} C_VEL
LIN {X 0,Y 355.798,Z 606.306,A -85,B 0,C 180,E1 -13651.379,E2 -13651.379} C_VEL
LIN {X 0,Y 357.745,Z 594.495,A -85,B 0,C 180,E1 -13653.014,E2 -13653.014} C_VEL
LIN {X 0,Y 359.703,Z 582.223,A -85,B 0,C 180,E1 -13654.413,E2 -13654.413} C_VEL
LIN {X 0,Y 361.564,Z 569.154,A -85,B 0,C 180,E1 -13655.634,E2 -13655.634} C_VEL
LIN {X 0,Y 363.014,Z 556.274,A -85,B 0,C 180,E1 -13656.616,E2 -13656.616} C_VEL
LIN {X 0,Y 364.443,Z 541.344,A -85,B 0,C 180,E1 -13657.502,E2 -13657.502} C_VEL
LIN {X 0,Y 365.534,Z 525.815,A -85,B 0,C 180,E1 -13658.176,E2 -13658.176} C_VEL
LIN {X 0,Y 366.239,Z 510.313,A -85,B 0,C 180,E1 -13658.616,E2 -13658.616} C_VEL
LIN {X 0,Y 370.172,Z 397.555,A -85,B 0,C 180,E1 -13661.061,E2 -13661.061} C_VEL
LIN {X 0,Y 363.47,Z 383.695,A -85,B 0,C 180,E1 -13662.183,E2 -13662.183} C_VEL
LIN {X 0,Y 356.781,Z 371.908,A -85,B 0,C 180,E1 -13663.33,E2 -13663.33} C_VEL
LIN {X 0,Y 352.032,Z 364.439,A -85,B 0,C 180,E1 -13664.158,E2 -13664.158} C_VEL
LIN {X 0,Y 349.828,Z 360.912,A -85,B 0,C 180,E1 -13664.564,E2 -13664.564} C_VEL
LIN {X 0,Y 348.196,Z 358.27,A -85,B 0,C 180,E1 -13664.87,E2 -13664.87} C_VEL
LIN {X 0,Y 347.865,Z 356.78,A -85,B 0,C 180,E1 -13664.979,E2 -13664.979} C_VEL
LIN {X 0,Y 347.886,Z 356.778,A -85,B 0,C 180,E1 -13668.344,E2 -13668.344} C_VEL
LIN {X 0,Y 348.001,Z 356.764,A -85,B 0,C 180,E1 -13671.873,E2 -13671.873} C_VEL
LIN {X 0,Y 348.04,Z 356.757,A -85,B 0,C 180,E1 -13674.205,E2 -13674.205} C_VEL
LIN {X 0,Y 348.191,Z 356.737,A -85,B 0,C 180,E1 -13677.686,E2 -13677.686} C_VEL
LIN {X 0,Y 348.285,Z 356.725,A -85,B 0,C 180,E1 -13680,E2 -13680} C_VEL
LIN {X 0,Y 348.205,Z 356.733,A -85,B 0,C 180,E1 -13682.313,E2 -13682.313} C_VEL
LIN {X 0,Y 348.058,Z 356.751,A -85,B 0,C 180,E1 -13686.958,E2 -13686.958} C_VEL
LIN {X 0,Y 347.899,Z 356.769,A -85,B 0,C 180,E1 -13690.475,E2 -13690.475} C_VEL
LIN {X 0,Y 347.901,Z 356.773,A -85,B 0,C 180,E1 -13694.149,E2 -13694.149} C_VEL
LIN {X 0,Y 347.831,Z 356.777,A -85,B 0,C 180,E1 -13698.259,E2 -13698.259} C_VEL
LIN {X 0,Y 347.791,Z 356.783,A -85,B 0,C 180,E1 -13701.635,E2 -13701.635} C_VEL
LIN {X 0,Y 347.815,Z 356.782,A -85,B 0,C 180,E1 -13705.108,E2 -13705.108} C_VEL
LIN {X 0,Y 347.813,Z 356.783,A -85,B 0,C 180,E1 -13707.693,E2 -13707.693} C_VEL
LIN {X 0,Y 347.766,Z 356.788,A -85,B 0,C 180,E1 -13710.346,E2 -13710.346} C_VEL
LIN {X 0,Y 347.746,Z 356.793,A -85,B 0,C 180,E1 -13714.463,E2 -13714.463} C_VEL
LIN {X 0,Y 347.775,Z 356.792,A -85,B 0,C 180,E1 -13717.988,E2 -13717.988} C_VEL
LIN {X 0,Y 347.752,Z 356.794,A -85,B 0,C 180,E1 -13721.83,E2 -13721.83} C_VEL
LIN {X 0,Y 347.767,Z 356.791,A -85,B 0,C 180,E1 -13725.016,E2 -13725.016} C_VEL
LIN {X 0,Y 347.753,Z 356.904,A -85,B 0,C 180,E1 -13728.727,E2 -13728.727} C_VEL
LIN {X 0,Y 350.958,Z 366.843,A -85,B 0,C 180,E1 -13731.626,E2 -13731.626} C_VEL
LIN {X 0,Y 354.03,Z 377.635,A -85,B 0,C 180,E1 -13734.479,E2 -13734.479} C_VEL
LIN {X 0,Y 355.719,Z 384.366,A -85,B 0,C 180,E1 -13736.078,E2 -13736.078} C_VEL
LIN {X 0,Y 362.334,Z 398.492,A -85,B 0,C 180,E1 -13737.272,E2 -13737.272} C_VEL
LIN {X 0,Y 363.537,Z 402.021,A -85,B 0,C 180,E1 -13737.507,E2 -13737.507} C_VEL
LIN {X 0,Y 367.428,Z 424.484,A -85,B 0,C 180,E1 -13738.53,E2 -13738.53} C_VEL
LIN {X 0,Y 369.16,Z 436.878,A -85,B 0,C 180,E1 -13739.033,E2 -13739.033} C_VEL
LIN {X 0,Y 365.058,Z 552.844,A -85,B 0,C 180,E1 -13741.544,E2 -13741.544} C_VEL
LIN {X 0,Y 363.933,Z 568.362,A -85,B 0,C 180,E1 -13742.076,E2 -13742.076} C_VEL
LIN {X 0,Y 362.343,Z 583.435,A -85,B 0,C 180,E1 -13742.805,E2 -13742.805} C_VEL
LIN {X 0,Y 360.608,Z 597.394,A -85,B 0,C 180,E1 -13743.702,E2 -13743.702} C_VEL
LIN {X 0,Y 358.509,Z 612.196,A -85,B 0,C 180,E1 -13744.917,E2 -13744.917} C_VEL
LIN {X 0,Y 356.365,Z 625.765,A -85,B 0,C 180,E1 -13746.307,E2 -13746.307} C_VEL
LIN {X 0,Y 354.228,Z 638.189,A -85,B 0,C 180,E1 -13747.854,E2 -13747.854} C_VEL
LIN {X 0,Y 352.282,Z 650.089,A -85,B 0,C 180,E1 -13749.659,E2 -13749.659} C_VEL
LIN {X 0,Y 350.539,Z 660.661,A -85,B 0,C 180,E1 -13751.592,E2 -13751.592} C_VEL
LIN {X 0,Y 348.968,Z 669.918,A -85,B 0,C 180,E1 -13753.623,E2 -13753.623} C_VEL
LIN {X 0,Y 347.725,Z 678.635,A -85,B 0,C 180,E1 -13755.963,E2 -13755.963} C_VEL
LIN {X 0,Y 346.929,Z 685.687,A -85,B 0,C 180,E1 -13758.312,E2 -13758.312} C_VEL
LIN {X 0,Y 346.427,Z 691.253,A -85,B 0,C 180,E1 -13760.659,E2 -13760.659} C_VEL
LIN {X 0,Y 346.292,Z 695.446,A -85,B 0,C 180,E1 -13763.005,E2 -13763.005} C_VEL
LIN {X 0,Y 346.217,Z 698.357,A -85,B 0,C 180,E1 -13765.342,E2 -13765.342} C_VEL
LIN {X 0,Y 346.288,Z 700.061,A -85,B 0,C 180,E1 -13767.673,E2 -13767.673} C_VEL
LIN {X 0,Y 346.389,Z 700.58,A -85,B 0,C 180,E1 -13769.999,E2 -13769.999} C_VEL
LIN {X 0,Y 346.307,Z 699.9,A -85,B 0,C 180,E1 -13772.326,E2 -13772.326} C_VEL
LIN {X 0,Y 346.231,Z 697.976,A -85,B 0,C 180,E1 -13774.657,E2 -13774.657} C_VEL
LIN {X 0,Y 346.296,Z 694.791,A -85,B 0,C 180,E1 -13776.994,E2 -13776.994} C_VEL
LIN {X 0,Y 346.42,Z 690.285,A -85,B 0,C 180,E1 -13779.34,E2 -13779.34} C_VEL
LIN {X 0,Y 346.926,Z 684.361,A -85,B 0,C 180,E1 -13781.687,E2 -13781.687} C_VEL
LIN {X 0,Y 347.689,Z 676.849,A -85,B 0,C 180,E1 -13784.037,E2 -13784.037} C_VEL
LIN {X 0,Y 348.7,Z 668.79,A -85,B 0,C 180,E1 -13786.088,E2 -13786.088} C_VEL
LIN {X 0,Y 350.135,Z 659.103,A -85,B 0,C 180,E1 -13788.126,E2 -13788.126} C_VEL
LIN {X 0,Y 351.708,Z 647.835,A -85,B 0,C 180,E1 -13790.087,E2 -13790.087} C_VEL
LIN {X 0,Y 353.465,Z 636.359,A -85,B 0,C 180,E1 -13791.735,E2 -13791.735} C_VEL
LIN {X 0,Y 355.01,Z 625.792,A -85,B 0,C 180,E1 -13793.015,E2 -13793.015} C_VEL
LIN {X 0,Y 356.533,Z 614.779,A -85,B 0,C 180,E1 -13794.143,E2 -13794.143} C_VEL
LIN {X 0,Y 358.23,Z 601.553,A -85,B 0,C 180,E1 -13795.258,E2 -13795.258} C_VEL
LIN {X 0,Y 359.799,Z 587.265,A -85,B 0,C 180,E1 -13796.22,E2 -13796.22} C_VEL
LIN {X 0,Y 361.175,Z 572.422,A -85,B 0,C 180,E1 -13796.976,E2 -13796.976} C_VEL
LIN {X 0,Y 362.208,Z 557.455,A -85,B 0,C 180,E1 -13797.518,E2 -13797.518} C_VEL
LIN {X 0,Y 363.065,Z 532.971,A -85,B 0,C 180,E1 -13798.074,E2 -13798.074} C_VEL
LIN {X 0,Y 365.895,Z 436.346,A -85,B 0,C 180,E1 -13800.1,E2 -13800.1} C_VEL
LIN {X 0,Y 360.602,Z 403.886,A -85,B 0,C 180,E1 -13801.316,E2 -13801.316} C_VEL
LIN {X 0,Y 358.794,Z 394.93,A -85,B 0,C 180,E1 -13801.689,E2 -13801.689} C_VEL
LIN {X 0,Y 355.742,Z 387.503,A -85,B 0,C 180,E1 -13802.158,E2 -13802.158} C_VEL
LIN {X 0,Y 352.399,Z 373.854,A -85,B 0,C 180,E1 -13805.148,E2 -13805.148} C_VEL
LIN {X 0,Y 348.831,Z 360.684,A -85,B 0,C 180,E1 -13808.211,E2 -13808.211} C_VEL
LIN {X 0,Y 347.771,Z 356.793,A -85,B 0,C 180,E1 -13809.16,E2 -13809.16} C_VEL
LIN {X 0,Y 347.748,Z 356.792,A -85,B 0,C 180,E1 -13811.83,E2 -13811.83} C_VEL
LIN {X 0,Y 347.763,Z 356.792,A -85,B 0,C 180,E1 -13815.016,E2 -13815.016} C_VEL
LIN {X 0,Y 347.747,Z 356.789,A -85,B 0,C 180,E1 -13818.397,E2 -13818.397} C_VEL
LIN {X 0,Y 347.771,Z 356.786,A -85,B 0,C 180,E1 -13822.011,E2 -13822.011} C_VEL
LIN {X 0,Y 347.741,Z 356.792,A -85,B 0,C 180,E1 -13825.536,E2 -13825.536} C_VEL
LIN {X 0,Y 347.76,Z 356.79,A -85,B 0,C 180,E1 -13829.654,E2 -13829.654} C_VEL
LIN {X 0,Y 347.848,Z 356.78,A -85,B 0,C 180,E1 -13832.745,E2 -13832.745} C_VEL
LIN {X 0,Y 347.785,Z 356.785,A -85,B 0,C 180,E1 -13836.162,E2 -13836.162} C_VEL
LIN {X 0,Y 347.809,Z 356.782,A -85,B 0,C 180,E1 -13839.91,E2 -13839.91} C_VEL
LIN {X 0,Y 347.863,Z 356.775,A -85,B 0,C 180,E1 -13842.359,E2 -13842.359} C_VEL
LIN {X 0,Y 347.894,Z 356.771,A -85,B 0,C 180,E1 -13845.971,E2 -13845.971} C_VEL
LIN {X 0,Y 347.926,Z 356.766,A -85,B 0,C 180,E1 -13849.526,E2 -13849.526} C_VEL
LIN {X 0,Y 348.089,Z 356.753,A -85,B 0,C 180,E1 -13853.042,E2 -13853.042} C_VEL
LIN {X 0,Y 348.206,Z 356.731,A -85,B 0,C 180,E1 -13857.687,E2 -13857.687} C_VEL
LIN {X 0,Y 348.344,Z 356.714,A -85,B 0,C 180,E1 -13860,E2 -13860} C_VEL
LIN {X 0,Y 348.205,Z 356.734,A -85,B 0,C 180,E1 -13862.314,E2 -13862.314} C_VEL
LIN {X 0,Y 348.104,Z 356.748,A -85,B 0,C 180,E1 -13866.958,E2 -13866.958} C_VEL
LIN {X 0,Y 347.965,Z 356.764,A -85,B 0,C 180,E1 -13869.299,E2 -13869.299} C_VEL
LIN {X 0,Y 347.888,Z 356.778,A -85,B 0,C 180,E1 -13872.84,E2 -13872.84} C_VEL
LIN {X 0,Y 347.837,Z 356.779,A -85,B 0,C 180,E1 -13876.432,E2 -13876.432} C_VEL
LIN {X 0,Y 347.853,Z 356.782,A -85,B 0,C 180,E1 -13878.861,E2 -13878.861} C_VEL
LIN {X 0,Y 347.76,Z 356.793,A -85,B 0,C 180,E1 -13882.581,E2 -13882.581} C_VEL
LIN {X 0,Y 347.809,Z 356.781,A -85,B 0,C 180,E1 -13885.109,E2 -13885.109} C_VEL
LIN {X 0,Y 347.809,Z 356.781,A -85,B 0,C 180,E1 -13887.695,E2 -13887.695} C_VEL
LIN {X 0,Y 347.763,Z 356.79,A -85,B 0,C 180,E1 -13890.347,E2 -13890.347} C_VEL
LIN {X 0,Y 347.743,Z 356.793,A -85,B 0,C 180,E1 -13894.465,E2 -13894.465} C_VEL
LIN {X 0,Y 347.772,Z 356.787,A -85,B 0,C 180,E1 -13897.989,E2 -13897.989} C_VEL
LIN {X 0,Y 347.749,Z 356.789,A -85,B 0,C 180,E1 -13901.831,E2 -13901.831} C_VEL
LIN {X 0,Y 347.705,Z 356.796,A -85,B 0,C 180,E1 -13905.028,E2 -13905.028} C_VEL
LIN {X 0,Y 347.747,Z 356.794,A -85,B 0,C 180,E1 -13908.399,E2 -13908.399} C_VEL
LIN {X 0,Y 347.772,Z 356.786,A -85,B 0,C 180,E1 -13912.013,E2 -13912.013} C_VEL
LIN {X 0,Y 347.745,Z 356.79,A -85,B 0,C 180,E1 -13915.537,E2 -13915.537} C_VEL
LIN {X 0,Y 347.746,Z 356.793,A -85,B 0,C 180,E1 -13918.301,E2 -13918.301} C_VEL
LIN {X 0,Y 347.748,Z 356.791,A -85,B 0,C 180,E1 -13920.986,E2 -13920.986} C_VEL
LIN {X 0,Y 347.76,Z 356.787,A -85,B 0,C 180,E1 -13923.603,E2 -13923.603} C_VEL
LIN {X 0,Y 347.778,Z 356.789,A -85,B 0,C 180,E1 -13926.162,E2 -13926.162} C_VEL
LIN {X 0,Y 347.788,Z 356.785,A -85,B 0,C 180,E1 -13929.908,E2 -13929.908} C_VEL
LIN {X 0,Y 347.8,Z 356.783,A -85,B 0,C 180,E1 -13933.567,E2 -13933.567} C_VEL
LIN {X 0,Y 347.89,Z 356.772,A -85,B 0,C 180,E1 -13937.161,E2 -13937.161} C_VEL
LIN {X 0,Y 347.938,Z 356.768,A -85,B 0,C 180,E1 -13940.701,E2 -13940.701} C_VEL
LIN {X 0,Y 348.043,Z 356.759,A -85,B 0,C 180,E1 -13944.206,E2 -13944.206} C_VEL
LIN {X 0,Y 348.192,Z 356.735,A -85,B 0,C 180,E1 -13947.687,E2 -13947.687} C_VEL
LIN {X 0,Y 348.135,Z 356.742,A -85,B 0,C 180,E1 -13951.157,E2 -13951.157} C_VEL
LIN {X 0,Y 348.191,Z 356.738,A -85,B 0,C 180,E1 -13952.314,E2 -13952.314} C_VEL
LIN {X 0,Y 348.065,Z 356.754,A -85,B 0,C 180,E1 -13956.959,E2 -13956.959} C_VEL
LIN {X 0,Y 348.044,Z 356.758,A -85,B 0,C 180,E1 -13957.36,E2 -13957.36} C_VEL
LIN {X 0,Y 349.138,Z 359.765,A -85,B 0,C 180,E1 -13957.555,E2 -13957.555} C_VEL
LIN {X 0,Y 362.436,Z 385.726,A -85,B 0,C 180,E1 -13959.391,E2 -13959.391} C_VEL
LIN {X 0,Y 366.445,Z 394.533,A -85,B 0,C 180,E1 -13959.94,E2 -13959.94} C_VEL
LIN {X 0,Y 364.409,Z 463.356,A -85,B 0,C 180,E1 -13961.384,E2 -13961.384} C_VEL
LIN {X 0,Y 362.925,Z 516.96,A -85,B 0,C 180,E1 -13962.548,E2 -13962.548} C_VEL
LIN {X 0,Y 362.114,Z 532.17,A -85,B 0,C 180,E1 -13963.093,E2 -13963.093} C_VEL
LIN {X 0,Y 360.965,Z 547.624,A -85,B 0,C 180,E1 -13963.887,E2 -13963.887} C_VEL
LIN {X 0,Y 359.551,Z 562.108,A -85,B 0,C 180,E1 -13964.866,E2 -13964.866} C_VEL
LIN {X 0,Y 358.156,Z 574.85,A -85,B 0,C 180,E1 -13965.946,E2 -13965.946} C_VEL
LIN {X 0,Y 356.369,Z 588.401,A -85,B 0,C 180,E1 -13967.355,E2 -13967.355} C_VEL
LIN {X 0,Y 354.596,Z 600.844,A -85,B 0,C 180,E1 -13968.939,E2 -13968.939} C_VEL
LIN {X 0,Y 352.926,Z 611.822,A -85,B 0,C 180,E1 -13970.619,E2 -13970.619} C_VEL
LIN {X 0,Y 351.287,Z 622.626,A -85,B 0,C 180,E1 -13972.622,E2 -13972.622} C_VEL
LIN {X 0,Y 350.104,Z 630.162,A -85,B 0,C 180,E1 -13974.29,E2 -13974.29} C_VEL
LIN {X 0,Y 349.01,Z 633.478,A -85,B 0,C 180,E1 -13975.07,E2 -13975.07} C_VEL
LIN {X 0,Y 345.439,Z 638.591,A -85,B 0,C 180,E1 -13976.342,E2 -13976.342} C_VEL
LIN {X 0,Y 341.891,Z 643.263,A -85,B 0,C 180,E1 -13977.685,E2 -13977.685} C_VEL
LIN {X 0,Y 340.855,Z 645.775,A -85,B 0,C 180,E1 -13978.565,E2 -13978.565} C_VEL
LIN {X 0,Y 340.272,Z 650.347,A -85,B 0,C 180,E1 -13980.443,E2 -13980.443} C_VEL
LIN {X 0,Y 339.772,Z 654.426,A -85,B 0,C 180,E1 -13982.534,E2 -13982.534} C_VEL
LIN {X 0,Y 339.429,Z 656.779,A -85,B 0,C 180,E1 -13984.083,E2 -13984.083} C_VEL
LIN {X 0,Y 339.135,Z 659.037,A -85,B 0,C 180,E1 -13986.078,E2 -13986.078} C_VEL
LIN {X 0,Y 339,Z 660.659,A -85,B 0,C 180,E1 -13988.459,E2 -13988.459} C_VEL
LIN {X 0,Y 339,Z 661.1,A -85,B 0,C 180,E1 -13989.992,E2 -13989.992} C_VEL
LIN {X 0,Y 339.022,Z 661.055,A -85,B 0,C 180,E1 -13991.729,E2 -13991.729} C_VEL
LIN {X 0,Y 339.177,Z 660.303,A -85,B 0,C 180,E1 -13993.512,E2 -13993.512} C_VEL
LIN {X 0,Y 339.435,Z 658.975,A -85,B 0,C 180,E1 -13995.253,E2 -13995.253} C_VEL
LIN {X 0,Y 339.771,Z 657.103,A -85,B 0,C 180,E1 -13996.953,E2 -13996.953} C_VEL
LIN {X 0,Y 340.347,Z 653.511,A -85,B 0,C 180,E1 -13999.251,E2 -13999.251} C_VEL
LIN {X 0,Y 341.271,Z 648.037,A -85,B 0,C 180,E1 -14001.843,E2 -14001.843} C_VEL
LIN {X 0,Y 342.495,Z 641.511,A -85,B 0,C 180,E1 -14004.209,E2 -14004.209} C_VEL
LIN {X 0,Y 344.077,Z 633.478,A -85,B 0,C 180,E1 -14006.53,E2 -14006.53} C_VEL
LIN {X 0,Y 345.91,Z 624.116,A -85,B 0,C 180,E1 -14008.723,E2 -14008.723} C_VEL
LIN {X 0,Y 348.016,Z 613.725,A -85,B 0,C 180,E1 -14010.713,E2 -14010.713} C_VEL
LIN {X 0,Y 350.078,Z 602.448,A -85,B 0,C 180,E1 -14012.5,E2 -14012.5} C_VEL
LIN {X 0,Y 352.19,Z 590.148,A -85,B 0,C 180,E1 -14014.107,E2 -14014.107} C_VEL
LIN {X 0,Y 354.271,Z 577.129,A -85,B 0,C 180,E1 -14015.493,E2 -14015.493} C_VEL
LIN {X 0,Y 355.945,Z 564.447,A -85,B 0,C 180,E1 -14016.599,E2 -14016.599} C_VEL
LIN {X 0,Y 357.655,Z 549.454,A -85,B 0,C 180,E1 -14017.636,E2 -14017.636} C_VEL
LIN {X 0,Y 358.948,Z 534.06,A -85,B 0,C 180,E1 -14018.443,E2 -14018.443} C_VEL
LIN {X 0,Y 359.894,Z 518.526,A -85,B 0,C 180,E1 -14019.009,E2 -14019.009} C_VEL
LIN {X 0,Y 364.266,Z 399.66,A -85,B 0,C 180,E1 -14021.662,E2 -14021.662} C_VEL
LIN {X 0,Y 357.501,Z 385.775,A -85,B 0,C 180,E1 -14022.849,E2 -14022.849} C_VEL
LIN {X 0,Y 349.955,Z 372.926,A -85,B 0,C 180,E1 -14024.189,E2 -14024.189} C_VEL
LIN {X 0,Y 344.9,Z 365.081,A -85,B 0,C 180,E1 -14025.13,E2 -14025.13} C_VEL
LIN {X 0,Y 343,Z 361.92,A -85,B 0,C 180,E1 -14025.501,E2 -14025.501} C_VEL
LIN {X 0,Y 341.364,Z 359.552,A -85,B 0,C 180,E1 -14025.821,E2 -14025.821} C_VEL
LIN {X 0,Y 340.876,Z 357.65,A -85,B 0,C 180,E1 -14025.969,E2 -14025.969} C_VEL
LIN {X 0,Y 340.851,Z 357.651,A -85,B 0,C 180,E1 -14029.305,E2 -14029.305} C_VEL
LIN {X 0,Y 341.003,Z 357.631,A -85,B 0,C 180,E1 -14032.896,E2 -14032.896} C_VEL
LIN {X 0,Y 340.815,Z 357.654,A -85,B 0,C 180,E1 -14035.268,E2 -14035.268} C_VEL
LIN {X 0,Y 341.128,Z 357.616,A -85,B 0,C 180,E1 -14037.638,E2 -14037.638} C_VEL
LIN {X 0,Y 341.237,Z 357.603,A -85,B 0,C 180,E1 -14040,E2 -14040} C_VEL
LIN {X 0,Y 341.167,Z 357.61,A -85,B 0,C 180,E1 -14042.361,E2 -14042.361} C_VEL
LIN {X 0,Y 341.005,Z 357.629,A -85,B 0,C 180,E1 -14047.103,E2 -14047.103} C_VEL
LIN {X 0,Y 340.851,Z 357.648,A -85,B 0,C 180,E1 -14050.694,E2 -14050.694} C_VEL
LIN {X 0,Y 340.866,Z 357.649,A -85,B 0,C 180,E1 -14054.324,E2 -14054.324} C_VEL
LIN {X 0,Y 340.788,Z 357.654,A -85,B 0,C 180,E1 -14058.44,E2 -14058.44} C_VEL
LIN {X 0,Y 340.756,Z 357.659,A -85,B 0,C 180,E1 -14061.856,E2 -14061.856} C_VEL
LIN {X 0,Y 340.775,Z 357.663,A -85,B 0,C 180,E1 -14065.664,E2 -14065.664} C_VEL
LIN {X 0,Y 340.743,Z 357.665,A -85,B 0,C 180,E1 -14068.319,E2 -14068.319} C_VEL
LIN {X 0,Y 340.706,Z 357.672,A -85,B 0,C 180,E1 -14071.043,E2 -14071.043} C_VEL
LIN {X 0,Y 340.719,Z 357.668,A -85,B 0,C 180,E1 -14075.278,E2 -14075.278} C_VEL
LIN {X 0,Y 340.711,Z 357.673,A -85,B 0,C 180,E1 -14078.386,E2 -14078.386} C_VEL
LIN {X 0,Y 340.7,Z 357.673,A -85,B 0,C 180,E1 -14082.045,E2 -14082.045} C_VEL
LIN {X 0,Y 340.685,Z 357.675,A -85,B 0,C 180,E1 -14085.461,E2 -14085.461} C_VEL
LIN {X 0,Y 340.7,Z 357.802,A -85,B 0,C 180,E1 -14087.803,E2 -14087.803} C_VEL
LIN {X 0,Y 344.043,Z 367.972,A -85,B 0,C 180,E1 -14090.918,E2 -14090.918} C_VEL
LIN {X 0,Y 347.333,Z 379.458,A -85,B 0,C 180,E1 -14094.07,E2 -14094.07} C_VEL
LIN {X 0,Y 348.399,Z 383.637,A -85,B 0,C 180,E1 -14095.102,E2 -14095.102} C_VEL
LIN {X 0,Y 356.047,Z 399.619,A -85,B 0,C 180,E1 -14096.547,E2 -14096.547} C_VEL
LIN {X 0,Y 357.942,Z 404.186,A -85,B 0,C 180,E1 -14096.908,E2 -14096.908} C_VEL
LIN {X 0,Y 361.636,Z 426.145,A -85,B 0,C 180,E1 -14097.935,E2 -14097.935} C_VEL
LIN {X 0,Y 363.249,Z 437.443,A -85,B 0,C 180,E1 -14098.411,E2 -14098.411} C_VEL
LIN {X 0,Y 358.95,Z 553.033,A -85,B 0,C 180,E1 -14100.974,E2 -14100.974} C_VEL
LIN {X 0,Y 357.795,Z 568.328,A -85,B 0,C 180,E1 -14101.513,E2 -14101.513} C_VEL
LIN {X 0,Y 356.078,Z 583.849,A -85,B 0,C 180,E1 -14102.285,E2 -14102.285} C_VEL
LIN {X 0,Y 354.157,Z 598.401,A -85,B 0,C 180,E1 -14103.251,E2 -14103.251} C_VEL
LIN {X 0,Y 352.088,Z 612.299,A -85,B 0,C 180,E1 -14104.427,E2 -14104.427} C_VEL
LIN {X 0,Y 349.852,Z 625.759,A -85,B 0,C 180,E1 -14105.838,E2 -14105.838} C_VEL
LIN {X 0,Y 347.599,Z 638.082,A -85,B 0,C 180,E1 -14107.408,E2 -14107.408} C_VEL
LIN {X 0,Y 345.699,Z 649.092,A -85,B 0,C 180,E1 -14109.105,E2 -14109.105} C_VEL
LIN {X 0,Y 343.995,Z 658.97,A -85,B 0,C 180,E1 -14110.919,E2 -14110.919} C_VEL
LIN {X 0,Y 342.267,Z 668.423,A -85,B 0,C 180,E1 -14112.986,E2 -14112.986} C_VEL
LIN {X 0,Y 341.052,Z 676.319,A -85,B 0,C 180,E1 -14115.073,E2 -14115.073} C_VEL
LIN {X 0,Y 340.055,Z 683.73,A -85,B 0,C 180,E1 -14117.466,E2 -14117.466} C_VEL
LIN {X 0,Y 339.447,Z 689.615,A -85,B 0,C 180,E1 -14119.863,E2 -14119.863} C_VEL
LIN {X 0,Y 339.264,Z 693.165,A -85,B 0,C 180,E1 -14121.662,E2 -14121.662} C_VEL
LIN {X 0,Y 339.168,Z 696.69,A -85,B 0,C 180,E1 -14124.053,E2 -14124.053} C_VEL
LIN {X 0,Y 339.133,Z 698.97,A -85,B 0,C 180,E1 -14126.435,E2 -14126.435} C_VEL
LIN {X 0,Y 339.301,Z 700.062,A -85,B 0,C 180,E1 -14128.813,E2 -14128.813} C_VEL
LIN {X 0,Y 339.319,Z 699.962,A -85,B 0,C 180,E1 -14131.186,E2 -14131.186} C_VEL
LIN {X 0,Y 339.141,Z 698.647,A -85,B 0,C 180,E1 -14133.564,E2 -14133.564} C_VEL
LIN {X 0,Y 339.167,Z 696.071,A -85,B 0,C 180,E1 -14135.946,E2 -14135.946} C_VEL
LIN {X 0,Y 339.26,Z 692.207,A -85,B 0,C 180,E1 -14138.337,E2 -14138.337} C_VEL
LIN {X 0,Y 339.54,Z 686.97,A -85,B 0,C 180,E1 -14140.736,E2 -14140.736} C_VEL
LIN {X 0,Y 340.248,Z 680.239,A -85,B 0,C 180,E1 -14143.132,E2 -14143.132} C_VEL
LIN {X 0,Y 341.166,Z 672.963,A -85,B 0,C 180,E1 -14145.227,E2 -14145.227} C_VEL
LIN {X 0,Y 342.328,Z 664.192,A -85,B 0,C 180,E1 -14147.318,E2 -14147.318} C_VEL
LIN {X 0,Y 343.779,Z 655.3,A -85,B 0,C 180,E1 -14149.092,E2 -14149.092} C_VEL
LIN {X 0,Y 345.421,Z 644.09,A -85,B 0,C 180,E1 -14150.967,E2 -14150.967} C_VEL
LIN {X 0,Y 347.186,Z 632.18,A -85,B 0,C 180,E1 -14152.619,E2 -14152.619} C_VEL
LIN {X 0,Y 349.103,Z 619.574,A -85,B 0,C 180,E1 -14154.058,E2 -14154.058} C_VEL
LIN {X 0,Y 351.113,Z 605.793,A -85,B 0,C 180,E1 -14155.331,E2 -14155.331} C_VEL
LIN {X 0,Y 352.894,Z 590.619,A -85,B 0,C 180,E1 -14156.445,E2 -14156.445} C_VEL
LIN {X 0,Y 354.373,Z 576.129,A -85,B 0,C 180,E1 -14157.258,E2 -14157.258} C_VEL
LIN {X 0,Y 355.561,Z 560.886,A -85,B 0,C 180,E1 -14157.877,E2 -14157.877} C_VEL
LIN {X 0,Y 356.314,Z 545.247,A -85,B 0,C 180,E1 -14158.293,E2 -14158.293} C_VEL
LIN {X 0,Y 359.573,Z 437.832,A -85,B 0,C 180,E1 -14160.585,E2 -14160.585} C_VEL
LIN {X 0,Y 355.344,Z 411.007,A -85,B 0,C 180,E1 -14161.597,E2 -14161.597} C_VEL
LIN {X 0,Y 352.79,Z 397.587,A -85,B 0,C 180,E1 -14162.155,E2 -14162.155} C_VEL
LIN {X 0,Y 348.405,Z 387.032,A -85,B 0,C 180,E1 -14162.85,E2 -14162.85} C_VEL
LIN {X 0,Y 345.158,Z 373.969,A -85,B 0,C 180,E1 -14165.794,E2 -14165.794} C_VEL
LIN {X 0,Y 341.266,Z 359.594,A -85,B 0,C 180,E1 -14169.239,E2 -14169.239} C_VEL
LIN {X 0,Y 340.7,Z 357.673,A -85,B 0,C 180,E1 -14169.752,E2 -14169.752} C_VEL
LIN {X 0,Y 340.674,Z 357.675,A -85,B 0,C 180,E1 -14172.904,E2 -14172.904} C_VEL
LIN {X 0,Y 340.664,Z 357.673,A -85,B 0,C 180,E1 -14176.224,E2 -14176.224} C_VEL
LIN {X 0,Y 340.685,Z 357.671,A -85,B 0,C 180,E1 -14179.753,E2 -14179.753} C_VEL
LIN {X 0,Y 340.702,Z 357.674,A -85,B 0,C 180,E1 -14183.258,E2 -14183.258} C_VEL
LIN {X 0,Y 340.688,Z 357.668,A -85,B 0,C 180,E1 -14186.153,E2 -14186.153} C_VEL
LIN {X 0,Y 340.771,Z 357.66,A -85,B 0,C 180,E1 -14190.333,E2 -14190.333} C_VEL
LIN {X 0,Y 340.801,Z 357.661,A -85,B 0,C 180,E1 -14193.02,E2 -14193.02} C_VEL
LIN {X 0,Y 340.725,Z 357.669,A -85,B 0,C 180,E1 -14196.927,E2 -14196.927} C_VEL
LIN {X 0,Y 340.787,Z 357.66,A -85,B 0,C 180,E1 -14200.734,E2 -14200.734} C_VEL
LIN {X 0,Y 340.784,Z 357.662,A -85,B 0,C 180,E1 -14203.219,E2 -14203.219} C_VEL
LIN {X 0,Y 340.841,Z 357.654,A -85,B 0,C 180,E1 -14206.891,E2 -14206.891} C_VEL
LIN {X 0,Y 340.923,Z 357.637,A -85,B 0,C 180,E1 -14210.508,E2 -14210.508} C_VEL
LIN {X 0,Y 341.057,Z 357.627,A -85,B 0,C 180,E1 -14212.898,E2 -14212.898} C_VEL
LIN {X 0,Y 341.167,Z 357.607,A -85,B 0,C 180,E1 -14217.639,E2 -14217.639} C_VEL
LIN {X 0,Y 341.294,Z 357.592,A -85,B 0,C 180,E1 -14220,E2 -14220} C_VEL
LIN {X 0,Y 341.167,Z 357.611,A -85,B 0,C 180,E1 -14222.362,E2 -14222.362} C_VEL
LIN {X 0,Y 341.074,Z 357.622,A -85,B 0,C 180,E1 -14227.102,E2 -14227.102} C_VEL
LIN {X 0,Y 340.869,Z 357.651,A -85,B 0,C 180,E1 -14230.694,E2 -14230.694} C_VEL
LIN {X 0,Y 340.861,Z 357.648,A -85,B 0,C 180,E1 -14234.325,E2 -14234.325} C_VEL
LIN {X 0,Y 340.836,Z 357.651,A -85,B 0,C 180,E1 -14238.468,E2 -14238.468} C_VEL
LIN {X 0,Y 340.716,Z 357.666,A -85,B 0,C 180,E1 -14241.842,E2 -14241.842} C_VEL
LIN {X 0,Y 340.77,Z 357.655,A -85,B 0,C 180,E1 -14245.665,E2 -14245.665} C_VEL
LIN {X 0,Y 340.74,Z 357.664,A -85,B 0,C 180,E1 -14248.32,E2 -14248.32} C_VEL
LIN {X 0,Y 340.703,Z 357.67,A -85,B 0,C 180,E1 -14251.045,E2 -14251.045} C_VEL
LIN {X 0,Y 340.717,Z 357.663,A -85,B 0,C 180,E1 -14255.28,E2 -14255.28} C_VEL
LIN {X 0,Y 340.708,Z 357.67,A -85,B 0,C 180,E1 -14258.387,E2 -14258.387} C_VEL
LIN {X 0,Y 340.698,Z 357.668,A -85,B 0,C 180,E1 -14262.046,E2 -14262.046} C_VEL
LIN {X 0,Y 340.652,Z 357.676,A -85,B 0,C 180,E1 -14266.228,E2 -14266.228} C_VEL
LIN {X 0,Y 340.685,Z 357.669,A -85,B 0,C 180,E1 -14269.755,E2 -14269.755} C_VEL
LIN {X 0,Y 340.705,Z 357.667,A -85,B 0,C 180,E1 -14273.259,E2 -14273.259} C_VEL
LIN {X 0,Y 340.694,Z 357.671,A -85,B 0,C 180,E1 -14276.154,E2 -14276.154} C_VEL
LIN {X 0,Y 340.725,Z 357.666,A -85,B 0,C 180,E1 -14280.035,E2 -14280.035} C_VEL
LIN {X 0,Y 340.727,Z 357.664,A -85,B 0,C 180,E1 -14283.014,E2 -14283.014} C_VEL
LIN {X 0,Y 340.758,Z 357.66,A -85,B 0,C 180,E1 -14285.639,E2 -14285.639} C_VEL
LIN {X 0,Y 340.73,Z 357.662,A -85,B 0,C 180,E1 -14289.474,E2 -14289.474} C_VEL
LIN {X 0,Y 340.764,Z 357.662,A -85,B 0,C 180,E1 -14291.98,E2 -14291.98} C_VEL
LIN {X 0,Y 340.835,Z 357.652,A -85,B 0,C 180,E1 -14295.731,E2 -14295.731} C_VEL
LIN {X 0,Y 340.851,Z 357.649,A -85,B 0,C 180,E1 -14299.306,E2 -14299.306} C_VEL
LIN {X 0,Y 341.005,Z 357.631,A -85,B 0,C 180,E1 -14302.897,E2 -14302.897} C_VEL
LIN {X 0,Y 340.816,Z 357.653,A -85,B 0,C 180,E1 -14305.269,E2 -14305.269} C_VEL
LIN {X 0,Y 341.129,Z 357.615,A -85,B 0,C 180,E1 -14307.639,E2 -14307.639} C_VEL
LIN {X 0,Y 341.104,Z 357.618,A -85,B 0,C 180,E1 -14311.181,E2 -14311.181} C_VEL
LIN {X 0,Y 341.128,Z 357.617,A -85,B 0,C 180,E1 -14312.362,E2 -14312.362} C_VEL
LIN {X 0,Y 341.017,Z 357.632,A -85,B 0,C 180,E1 -14316.695,E2 -14316.695} C_VEL
LIN {X 0,Y 342.098,Z 360.583,A -85,B 0,C 180,E1 -14316.896,E2 -14316.896} C_VEL
LIN {X 0,Y 352.376,Z 380.395,A -85,B 0,C 180,E1 -14318.378,E2 -14318.378} C_VEL
LIN {X 0,Y 359.801,Z 395.794,A -85,B 0,C 180,E1 -14319.411,E2 -14319.411} C_VEL
LIN {X 0,Y 360.247,Z 397.561,A -85,B 0,C 180,E1 -14319.491,E2 -14319.491} C_VEL
LIN {X 0,Y 356.529,Z 516.667,A -85,B 0,C 180,E1 -14322.054,E2 -14322.054} C_VEL
LIN {X 0,Y 355.721,Z 531.594,A -85,B 0,C 180,E1 -14322.586,E2 -14322.586} C_VEL
LIN {X 0,Y 354.514,Z 547.519,A -85,B 0,C 180,E1 -14323.405,E2 -14323.405} C_VEL
LIN {X 0,Y 353.053,Z 562.206,A -85,B 0,C 180,E1 -14324.409,E2 -14324.409} C_VEL
LIN {X 0,Y 351.484,Z 575.912,A -85,B 0,C 180,E1 -14325.596,E2 -14325.596} C_VEL
LIN {X 0,Y 349.756,Z 588.613,A -85,B 0,C 180,E1 -14326.94,E2 -14326.94} C_VEL
LIN {X 0,Y 347.868,Z 601.247,A -85,B 0,C 180,E1 -14328.572,E2 -14328.572} C_VEL
LIN {X 0,Y 346.201,Z 611.676,A -85,B 0,C 180,E1 -14330.189,E2 -14330.189} C_VEL
LIN {X 0,Y 344.528,Z 622.316,A -85,B 0,C 180,E1 -14332.172,E2 -14332.172} C_VEL
LIN {X 0,Y 343.113,Z 631.241,A -85,B 0,C 180,E1 -14334.184,E2 -14334.184} C_VEL
LIN {X 0,Y 341.863,Z 638.783,A -85,B 0,C 180,E1 -14336.232,E2 -14336.232} C_VEL
LIN {X 0,Y 340.855,Z 645.775,A -85,B 0,C 180,E1 -14338.565,E2 -14338.565} C_VEL
LIN {X 0,Y 339.88,Z 648.17,A -85,B 0,C 180,E1 -14339.46,E2 -14339.46} C_VEL
LIN {X 0,Y 335.174,Z 653.08,A -85,B 0,C 180,E1 -14341.519,E2 -14341.519} C_VEL
LIN {X 0,Y 332.94,Z 655.368,A -85,B 0,C 180,E1 -14342.767,E2 -14342.767} C_VEL
LIN {X 0,Y 332.471,Z 656.338,A -85,B 0,C 180,E1 -14343.423,E2 -14343.423} C_VEL
LIN {X 0,Y 332.2,Z 658.199,A -85,B 0,C 180,E1 -14344.835,E2 -14344.835} C_VEL
LIN {X 0,Y 332.017,Z 659.829,A -85,B 0,C 180,E1 -14346.45,E2 -14346.45} C_VEL
LIN {X 0,Y 331.926,Z 661.047,A -85,B 0,C 180,E1 -14348.425,E2 -14348.425} C_VEL
LIN {X 0,Y 331.904,Z 661.546,A -85,B 0,C 180,E1 -14351.028,E2 -14351.028} C_VEL
LIN {X 0,Y 332.005,Z 661.193,A -85,B 0,C 180,E1 -14352.64,E2 -14352.64} C_VEL
LIN {X 0,Y 332.208,Z 660.333,A -85,B 0,C 180,E1 -14354.278,E2 -14354.278} C_VEL
LIN {X 0,Y 332.474,Z 658.914,A -85,B 0,C 180,E1 -14355.949,E2 -14355.949} C_VEL
LIN {X 0,Y 333.049,Z 655.753,A -85,B 0,C 180,E1 -14358.416,E2 -14358.416} C_VEL
LIN {X 0,Y 333.944,Z 650.753,A -85,B 0,C 180,E1 -14361.141,E2 -14361.141} C_VEL
LIN {X 0,Y 335.029,Z 645.016,A -85,B 0,C 180,E1 -14363.498,E2 -14363.498} C_VEL
LIN {X 0,Y 336.386,Z 638.418,A -85,B 0,C 180,E1 -14365.659,E2 -14365.659} C_VEL
LIN {X 0,Y 338.074,Z 630.275,A -85,B 0,C 180,E1 -14367.848,E2 -14367.848} C_VEL
LIN {X 0,Y 340.088,Z 620.944,A -85,B 0,C 180,E1 -14369.903,E2 -14369.903} C_VEL
LIN {X 0,Y 342.182,Z 610.505,A -85,B 0,C 180,E1 -14371.81,E2 -14371.81} C_VEL
LIN {X 0,Y 344.406,Z 598.563,A -85,B 0,C 180,E1 -14373.612,E2 -14373.612} C_VEL
LIN {X 0,Y 346.528,Z 586.416,A -85,B 0,C 180,E1 -14375.117,E2 -14375.117} C_VEL
LIN {X 0,Y 348.498,Z 574.171,A -85,B 0,C 180,E1 -14376.367,E2 -14376.367} C_VEL
LIN {X 0,Y 350.329,Z 560.477,A -85,B 0,C 180,E1 -14377.51,E2 -14377.51} C_VEL
LIN {X 0,Y 351.98,Z 545.636,A -85,B 0,C 180,E1 -14378.475,E2 -14378.475} C_VEL
LIN {X 0,Y 353.18,Z 530.661,A -85,B 0,C 180,E1 -14379.209,E2 -14379.209} C_VEL
LIN {X 0,Y 354.035,Z 516.172,A -85,B 0,C 180,E1 -14379.696,E2 -14379.696} C_VEL
LIN {X 0,Y 358.488,Z 402.136,A -85,B 0,C 180,E1 -14382.272,E2 -14382.272} C_VEL
LIN {X 0,Y 352.92,Z 390.526,A -85,B 0,C 180,E1 -14383.291,E2 -14383.291} C_VEL
LIN {X 0,Y 345.996,Z 378.402,A -85,B 0,C 180,E1 -14384.571,E2 -14384.571} C_VEL
LIN {X 0,Y 338.339,Z 366.453,A -85,B 0,C 180,E1 -14386.061,E2 -14386.061} C_VEL
LIN {X 0,Y 336.124,Z 362.925,A -85,B 0,C 180,E1 -14386.519,E2 -14386.519} C_VEL
LIN {X 0,Y 334.416,Z 360.664,A -85,B 0,C 180,E1 -14386.865,E2 -14386.865} C_VEL
LIN {X 0,Y 333.793,Z 358.534,A -85,B 0,C 180,E1 -14387.073,E2 -14387.073} C_VEL
LIN {X 0,Y 333.823,Z 358.529,A -85,B 0,C 180,E1 -14390.303,E2 -14390.303} C_VEL
LIN {X 0,Y 333.989,Z 358.509,A -85,B 0,C 180,E1 -14393.96,E2 -14393.96} C_VEL
LIN {X 0,Y 334.069,Z 358.495,A -85,B 0,C 180,E1 -14397.588,E2 -14397.588} C_VEL
LIN {X 0,Y 334.19,Z 358.48,A -85,B 0,C 180,E1 -14400,E2 -14400} C_VEL
LIN {X 0,Y 334.104,Z 358.49,A -85,B 0,C 180,E1 -14402.411,E2 -14402.411} C_VEL
LIN {X 0,Y 333.994,Z 358.507,A -85,B 0,C 180,E1 -14406.039,E2 -14406.039} C_VEL
LIN {X 0,Y 333.823,Z 358.523,A -85,B 0,C 180,E1 -14409.696,E2 -14409.696} C_VEL
LIN {X 0,Y 333.799,Z 358.526,A -85,B 0,C 180,E1 -14413.391,E2 -14413.391} C_VEL
LIN {X 0,Y 333.722,Z 358.54,A -85,B 0,C 180,E1 -14417.147,E2 -14417.147} C_VEL
LIN {X 0,Y 333.724,Z 358.539,A -85,B 0,C 180,E1 -14419.691,E2 -14419.691} C_VEL
LIN {X 0,Y 333.695,Z 358.541,A -85,B 0,C 180,E1 -14422.278,E2 -14422.278} C_VEL
LIN {X 0,Y 333.738,Z 358.538,A -85,B 0,C 180,E1 -14426.246,E2 -14426.246} C_VEL
LIN {X 0,Y 333.713,Z 358.541,A -85,B 0,C 180,E1 -14428.971,E2 -14428.971} C_VEL
LIN {X 0,Y 333.645,Z 358.546,A -85,B 0,C 180,E1 -14432.586,E2 -14432.586} C_VEL
LIN {X 0,Y 333.677,Z 358.548,A -85,B 0,C 180,E1 -14436.138,E2 -14436.138} C_VEL
LIN {X 0,Y 333.648,Z 358.549,A -85,B 0,C 180,E1 -14439.192,E2 -14439.192} C_VEL
LIN {X 0,Y 333.634,Z 358.553,A -85,B 0,C 180,E1 -14442.5,E2 -14442.5} C_VEL
LIN {X 0,Y 333.624,Z 358.553,A -85,B 0,C 180,E1 -14445.959,E2 -14445.959} C_VEL
LIN {X 0,Y 333.635,Z 358.591,A -85,B 0,C 180,E1 -14446.776,E2 -14446.776} C_VEL
LIN {X 0,Y 336.962,Z 368.745,A -85,B 0,C 180,E1 -14450.046,E2 -14450.046} C_VEL
LIN {X 0,Y 339.803,Z 378.211,A -85,B 0,C 180,E1 -14452.795,E2 -14452.795} C_VEL
LIN {X 0,Y 341.153,Z 383.077,A -85,B 0,C 180,E1 -14454.069,E2 -14454.069} C_VEL
LIN {X 0,Y 348.397,Z 397.738,A -85,B 0,C 180,E1 -14455.52,E2 -14455.52} C_VEL
LIN {X 0,Y 352.511,Z 406.918,A -85,B 0,C 180,E1 -14456.31,E2 -14456.31} C_VEL
LIN {X 0,Y 356.179,Z 429.6,A -85,B 0,C 180,E1 -14457.397,E2 -14457.397} C_VEL
LIN {X 0,Y 357.398,Z 439.532,A -85,B 0,C 180,E1 -14457.811,E2 -14457.811} C_VEL
LIN {X 0,Y 352.981,Z 552.418,A -85,B 0,C 180,E1 -14460.353,E2 -14460.353} C_VEL
LIN {X 0,Y 351.777,Z 567.693,A -85,B 0,C 180,E1 -14460.898,E2 -14460.898} C_VEL
LIN {X 0,Y 349.965,Z 583.205,A -85,B 0,C 180,E1 -14461.677,E2 -14461.677} C_VEL
LIN {X 0,Y 347.945,Z 597.967,A -85,B 0,C 180,E1 -14462.673,E2 -14462.673} C_VEL
LIN {X 0,Y 345.7,Z 612.398,A -85,B 0,C 180,E1 -14463.919,E2 -14463.919} C_VEL
LIN {X 0,Y 343.346,Z 625.767,A -85,B 0,C 180,E1 -14465.35,E2 -14465.35} C_VEL
LIN {X 0,Y 341.011,Z 638.02,A -85,B 0,C 180,E1 -14466.947,E2 -14466.947} C_VEL
LIN {X 0,Y 338.957,Z 649.274,A -85,B 0,C 180,E1 -14468.725,E2 -14468.725} C_VEL
LIN {X 0,Y 337.188,Z 658.798,A -85,B 0,C 180,E1 -14470.519,E2 -14470.519} C_VEL
LIN {X 0,Y 335.42,Z 668.189,A -85,B 0,C 180,E1 -14472.627,E2 -14472.627} C_VEL
LIN {X 0,Y 333.943,Z 677.098,A -85,B 0,C 180,E1 -14475.059,E2 -14475.059} C_VEL
LIN {X 0,Y 333.039,Z 683.437,A -85,B 0,C 180,E1 -14477.198,E2 -14477.198} C_VEL
LIN {X 0,Y 332.395,Z 689.295,A -85,B 0,C 180,E1 -14479.646,E2 -14479.646} C_VEL
LIN {X 0,Y 332.196,Z 692.828,A -85,B 0,C 180,E1 -14481.483,E2 -14481.483} C_VEL
LIN {X 0,Y 332.074,Z 696.549,A -85,B 0,C 180,E1 -14484.1,E2 -14484.1} C_VEL
LIN {X 0,Y 332.055,Z 698.585,A -85,B 0,C 180,E1 -14486.359,E2 -14486.359} C_VEL
LIN {X 0,Y 332.206,Z 699.656,A -85,B 0,C 180,E1 -14488.787,E2 -14488.787} C_VEL
LIN {X 0,Y 332.239,Z 699.531,A -85,B 0,C 180,E1 -14491.212,E2 -14491.212} C_VEL
LIN {X 0,Y 332.063,Z 698.194,A -85,B 0,C 180,E1 -14493.64,E2 -14493.64} C_VEL
LIN {X 0,Y 332.094,Z 695.601,A -85,B 0,C 180,E1 -14496.073,E2 -14496.073} C_VEL
LIN {X 0,Y 332.192,Z 691.705,A -85,B 0,C 180,E1 -14498.516,E2 -14498.516} C_VEL
LIN {X 0,Y 332.502,Z 686.433,A -85,B 0,C 180,E1 -14500.966,E2 -14500.966} C_VEL
LIN {X 0,Y 333.226,Z 679.662,A -85,B 0,C 180,E1 -14503.414,E2 -14503.414} C_VEL
LIN {X 0,Y 334.198,Z 672.343,A -85,B 0,C 180,E1 -14505.552,E2 -14505.552} C_VEL
LIN {X 0,Y 335.452,Z 663.524,A -85,B 0,C 180,E1 -14507.685,E2 -14507.685} C_VEL
LIN {X 0,Y 336.939,Z 654.563,A -85,B 0,C 180,E1 -14509.495,E2 -14509.495} C_VEL
LIN {X 0,Y 338.562,Z 643.967,A -85,B 0,C 180,E1 -14511.301,E2 -14511.301} C_VEL
LIN {X 0,Y 340.369,Z 632.456,A -85,B 0,C 180,E1 -14512.937,E2 -14512.937} C_VEL
LIN {X 0,Y 342.345,Z 619.961,A -85,B 0,C 180,E1 -14514.402,E2 -14514.402} C_VEL
LIN {X 0,Y 344.368,Z 606.434,A -85,B 0,C 180,E1 -14515.692,E2 -14515.692} C_VEL
LIN {X 0,Y 346.228,Z 591.668,A -85,B 0,C 180,E1 -14516.816,E2 -14516.816} C_VEL
LIN {X 0,Y 347.805,Z 576.602,A -85,B 0,C 180,E1 -14517.694,E2 -14517.694} C_VEL
LIN {X 0,Y 349.093,Z 560.66,A -85,B 0,C 180,E1 -14518.358,E2 -14518.358} C_VEL
LIN {X 0,Y 349.883,Z 545.149,A -85,B 0,C 180,E1 -14518.78,E2 -14518.78} C_VEL
LIN {X 0,Y 353.25,Z 438.281,A -85,B 0,C 180,E1 -14521.101,E2 -14521.101} C_VEL
LIN {X 0,Y 348.933,Z 411.375,A -85,B 0,C 180,E1 -14522.153,E2 -14522.153} C_VEL
LIN {X 0,Y 346.721,Z 399.929,A -85,B 0,C 180,E1 -14522.647,E2 -14522.647} C_VEL
LIN {X 0,Y 341.062,Z 386.584,A -85,B 0,C 180,E1 -14523.559,E2 -14523.559} C_VEL
LIN {X 0,Y 337.639,Z 372.914,A -85,B 0,C 180,E1 -14526.739,E2 -14526.739} C_VEL
LIN {X 0,Y 333.646,Z 358.553,A -85,B 0,C 180,E1 -14530.322,E2 -14530.322} C_VEL
LIN {X 0,Y 333.618,Z 358.552,A -85,B 0,C 180,E1 -14534.041,E2 -14534.041} C_VEL
LIN {X 0,Y 333.639,Z 358.547,A -85,B 0,C 180,E1 -14537.618,E2 -14537.618} C_VEL
LIN {X 0,Y 333.649,Z 358.549,A -85,B 0,C 180,E1 -14541.202,E2 -14541.202} C_VEL
LIN {X 0,Y 333.673,Z 358.546,A -85,B 0,C 180,E1 -14543.861,E2 -14543.861} C_VEL
LIN {X 0,Y 333.64,Z 358.551,A -85,B 0,C 180,E1 -14547.413,E2 -14547.413} C_VEL
LIN {X 0,Y 333.707,Z 358.544,A -85,B 0,C 180,E1 -14551.028,E2 -14551.028} C_VEL
LIN {X 0,Y 333.732,Z 358.536,A -85,B 0,C 180,E1 -14553.754,E2 -14553.754} C_VEL
LIN {X 0,Y 333.716,Z 358.537,A -85,B 0,C 180,E1 -14557.914,E2 -14557.914} C_VEL
LIN {X 0,Y 333.79,Z 358.529,A -85,B 0,C 180,E1 -14561.59,E2 -14561.59} C_VEL
LIN {X 0,Y 333.805,Z 358.527,A -85,B 0,C 180,E1 -14565.577,E2 -14565.577} C_VEL
LIN {X 0,Y 333.831,Z 358.521,A -85,B 0,C 180,E1 -14569.078,E2 -14569.078} C_VEL
LIN {X 0,Y 334.009,Z 358.503,A -85,B 0,C 180,E1 -14572.748,E2 -14572.748} C_VEL
LIN {X 0,Y 333.807,Z 358.529,A -85,B 0,C 180,E1 -14575.169,E2 -14575.169} C_VEL
LIN {X 0,Y 334.104,Z 358.487,A -85,B 0,C 180,E1 -14577.589,E2 -14577.589} C_VEL
LIN {X 0,Y 334.245,Z 358.47,A -85,B 0,C 180,E1 -14580,E2 -14580} C_VEL
LIN {X 0,Y 334.104,Z 358.491,A -85,B 0,C 180,E1 -14582.412,E2 -14582.412} C_VEL
LIN {X 0,Y 334.023,Z 358.498,A -85,B 0,C 180,E1 -14587.253,E2 -14587.253} C_VEL
LIN {X 0,Y 333.832,Z 358.528,A -85,B 0,C 180,E1 -14590.922,E2 -14590.922} C_VEL
LIN {X 0,Y 333.806,Z 358.53,A -85,B 0,C 180,E1 -14594.635,E2 -14594.635} C_VEL
LIN {X 0,Y 333.795,Z 358.53,A -85,B 0,C 180,E1 -14598.656,E2 -14598.656} C_VEL
LIN {X 0,Y 333.655,Z 358.547,A -85,B 0,C 180,E1 -14602.281,E2 -14602.281} C_VEL
LIN {X 0,Y 333.734,Z 358.532,A -85,B 0,C 180,E1 -14606.247,E2 -14606.247} C_VEL
LIN {X 0,Y 333.71,Z 358.542,A -85,B 0,C 180,E1 -14608.973,E2 -14608.973} C_VEL
LIN {X 0,Y 333.642,Z 358.551,A -85,B 0,C 180,E1 -14612.588,E2 -14612.588} C_VEL
LIN {X 0,Y 333.675,Z 358.54,A -85,B 0,C 180,E1 -14616.14,E2 -14616.14} C_VEL
LIN {X 0,Y 333.646,Z 358.548,A -85,B 0,C 180,E1 -14619.193,E2 -14619.193} C_VEL
LIN {X 0,Y 333.632,Z 358.551,A -85,B 0,C 180,E1 -14622.501,E2 -14622.501} C_VEL
LIN {X 0,Y 333.596,Z 358.553,A -85,B 0,C 180,E1 -14625.956,E2 -14625.956} C_VEL
LIN {X 0,Y 333.646,Z 358.546,A -85,B 0,C 180,E1 -14629.317,E2 -14629.317} C_VEL
LIN {X 0,Y 333.665,Z 358.545,A -85,B 0,C 180,E1 -14633.169,E2 -14633.169} C_VEL
LIN {X 0,Y 333.675,Z 358.543,A -85,B 0,C 180,E1 -14635.342,E2 -14635.342} C_VEL
LIN {X 0,Y 333.631,Z 358.55,A -85,B 0,C 180,E1 -14638.223,E2 -14638.223} C_VEL
LIN {X 0,Y 333.657,Z 358.547,A -85,B 0,C 180,E1 -14641.023,E2 -14641.023} C_VEL
LIN {X 0,Y 333.711,Z 358.538,A -85,B 0,C 180,E1 -14645.09,E2 -14645.09} C_VEL
LIN {X 0,Y 333.671,Z 358.542,A -85,B 0,C 180,E1 -14649.019,E2 -14649.019} C_VEL
LIN {X 0,Y 333.688,Z 358.542,A -85,B 0,C 180,E1 -14652.851,E2 -14652.851} C_VEL
LIN {X 0,Y 333.79,Z 358.532,A -85,B 0,C 180,E1 -14656.609,E2 -14656.609} C_VEL
LIN {X 0,Y 333.824,Z 358.53,A -85,B 0,C 180,E1 -14660.304,E2 -14660.304} C_VEL
LIN {X 0,Y 333.992,Z 358.507,A -85,B 0,C 180,E1 -14663.961,E2 -14663.961} C_VEL
LIN {X 0,Y 334.07,Z 358.495,A -85,B 0,C 180,E1 -14667.589,E2 -14667.589} C_VEL
LIN {X 0,Y 334.074,Z 358.494,A -85,B 0,C 180,E1 -14671.206,E2 -14671.206} C_VEL
LIN {X 0,Y 334.068,Z 358.495,A -85,B 0,C 180,E1 -14672.412,E2 -14672.412} C_VEL
LIN {X 0,Y 333.975,Z 358.507,A -85,B 0,C 180,E1 -14676.002,E2 -14676.002} C_VEL
LIN {X 0,Y 335.005,Z 361.417,A -85,B 0,C 180,E1 -14676.207,E2 -14676.207} C_VEL
LIN {X 0,Y 343.004,Z 376.358,A -85,B 0,C 180,E1 -14677.395,E2 -14677.395} C_VEL
LIN {X 0,Y 353.904,Z 398.642,A -85,B 0,C 180,E1 -14678.969,E2 -14678.969} C_VEL
LIN {X 0,Y 350.098,Z 517.408,A -85,B 0,C 180,E1 -14681.581,E2 -14681.581} C_VEL
LIN {X 0,Y 349.26,Z 532.283,A -85,B 0,C 180,E1 -14682.125,E2 -14682.125} C_VEL
LIN {X 0,Y 348.032,Z 547.877,A -85,B 0,C 180,E1 -14682.942,E2 -14682.942} C_VEL
LIN {X 0,Y 346.559,Z 562.216,A -85,B 0,C 180,E1 -14683.934,E2 -14683.934} C_VEL
LIN {X 0,Y 344.839,Z 576.702,A -85,B 0,C 180,E1 -14685.213,E2 -14685.213} C_VEL
LIN {X 0,Y 343.159,Z 588.562,A -85,B 0,C 180,E1 -14686.486,E2 -14686.486} C_VEL
LIN {X 0,Y 341.394,Z 600.132,A -85,B 0,C 180,E1 -14687.987,E2 -14687.987} C_VEL
LIN {X 0,Y 339.647,Z 610.862,A -85,B 0,C 180,E1 -14689.649,E2 -14689.649} C_VEL
LIN {X 0,Y 338.07,Z 620.312,A -85,B 0,C 180,E1 -14691.386,E2 -14691.386} C_VEL
LIN {X 0,Y 336.533,Z 629.427,A -85,B 0,C 180,E1 -14693.378,E2 -14693.378} C_VEL
LIN {X 0,Y 335.14,Z 637.865,A -85,B 0,C 180,E1 -14695.613,E2 -14695.613} C_VEL
LIN {X 0,Y 334.021,Z 644.911,A -85,B 0,C 180,E1 -14697.906,E2 -14697.906} C_VEL
LIN {X 0,Y 333.199,Z 650.991,A -85,B 0,C 180,E1 -14700.413,E2 -14700.413} C_VEL
LIN {X 0,Y 332.725,Z 654.665,A -85,B 0,C 180,E1 -14702.338,E2 -14702.338} C_VEL
LIN {X 0,Y 332.471,Z 656.338,A -85,B 0,C 180,E1 -14703.423,E2 -14703.423} C_VEL
LIN {X 0,Y 331.588,Z 657.728,A -85,B 0,C 180,E1 -14704.406,E2 -14704.406} C_VEL
LIN {X 0,Y 328.463,Z 659.627,A -85,B 0,C 180,E1 -14706.009,E2 -14706.009} C_VEL
LIN {X 0,Y 325.939,Z 660.787,A -85,B 0,C 180,E1 -14707.317,E2 -14707.317} C_VEL
LIN {X 0,Y 324.894,Z 661.409,A -85,B 0,C 180,E1 -14708.338,E2 -14708.338} C_VEL
LIN {X 0,Y 324.824,Z 661.547,A -85,B 0,C 180,E1 -14708.685,E2 -14708.685} C_VEL
LIN {X 0,Y 324.815,Z 661.992,A -85,B 0,C 180,E1 -14710.773,E2 -14710.773} C_VEL
LIN {X 0,Y 324.934,Z 661.645,A -85,B 0,C 180,E1 -14712.659,E2 -14712.659} C_VEL
LIN {X 0,Y 325.149,Z 660.715,A -85,B 0,C 180,E1 -14714.496,E2 -14714.496} C_VEL
LIN {X 0,Y 325.672,Z 658.143,A -85,B 0,C 180,E1 -14717.2,E2 -14717.2} C_VEL
LIN {X 0,Y 326.383,Z 654.37,A -85,B 0,C 180,E1 -14719.759,E2 -14719.759} C_VEL
LIN {X 0,Y 327.27,Z 649.807,A -85,B 0,C 180,E1 -14722.057,E2 -14722.057} C_VEL
LIN {X 0,Y 328.503,Z 643.929,A -85,B 0,C 180,E1 -14724.388,E2 -14724.388} C_VEL
LIN {X 0,Y 330.145,Z 636.446,A -85,B 0,C 180,E1 -14726.759,E2 -14726.759} C_VEL
LIN {X 0,Y 331.859,Z 628.602,A -85,B 0,C 180,E1 -14728.799,E2 -14728.799} C_VEL
LIN {X 0,Y 333.972,Z 619.319,A -85,B 0,C 180,E1 -14730.795,E2 -14730.795} C_VEL
LIN {X 0,Y 336.094,Z 609.217,A -85,B 0,C 180,E1 -14732.61,E2 -14732.61} C_VEL
LIN {X 0,Y 338.263,Z 597.987,A -85,B 0,C 180,E1 -14734.296,E2 -14734.296} C_VEL
LIN {X 0,Y 340.468,Z 586.03,A -85,B 0,C 180,E1 -14735.778,E2 -14735.778} C_VEL
LIN {X 0,Y 342.717,Z 572.359,A -85,B 0,C 180,E1 -14737.164,E2 -14737.164} C_VEL
LIN {X 0,Y 344.601,Z 558.33,A -85,B 0,C 180,E1 -14738.305,E2 -14738.305} C_VEL
LIN {X 0,Y 346.256,Z 543.39,A -85,B 0,C 180,E1 -14739.245,E2 -14739.245} C_VEL
LIN {X 0,Y 347.494,Z 527.874,A -85,B 0,C 180,E1 -14739.967,E2 -14739.967} C_VEL
LIN {X 0,Y 348.342,Z 512.299,A -85,B 0,C 180,E1 -14740.44,E2 -14740.44} C_VEL
LIN {X 0,Y 352.786,Z 404.438,A -85,B 0,C 180,E1 -14742.911,E2 -14742.911} C_VEL
LIN {X 0,Y 347.563,Z 393.767,A -85,B 0,C 180,E1 -14743.894,E2 -14743.894} C_VEL
LIN {X 0,Y 341.136,Z 382.514,A -85,B 0,C 180,E1 -14745.135,E2 -14745.135} C_VEL
LIN {X 0,Y 333.698,Z 370.774,A -85,B 0,C 180,E1 -14746.647,E2 -14746.647} C_VEL
LIN {X 0,Y 331.843,Z 367.929,A -85,B 0,C 180,E1 -14747.042,E2 -14747.042} C_VEL
LIN {X 0,Y 329.847,Z 364.703,A -85,B 0,C 180,E1 -14747.486,E2 -14747.486} C_VEL
LIN {X 0,Y 327.457,Z 361.713,A -85,B 0,C 180,E1 -14747.999,E2 -14747.999} C_VEL
LIN {X 0,Y 326.762,Z 359.408,A -85,B 0,C 180,E1 -14748.209,E2 -14748.209} C_VEL
LIN {X 0,Y 326.915,Z 359.387,A -85,B 0,C 180,E1 -14752.588,E2 -14752.588} C_VEL
LIN {X 0,Y 326.75,Z 359.406,A -85,B 0,C 180,E1 -14755.064,E2 -14755.064} C_VEL
LIN {X 0,Y 327.012,Z 359.374,A -85,B 0,C 180,E1 -14757.536,E2 -14757.536} C_VEL
LIN {X 0,Y 327.143,Z 359.358,A -85,B 0,C 180,E1 -14760,E2 -14760} C_VEL
LIN {X 0,Y 327.044,Z 359.369,A -85,B 0,C 180,E1 -14762.463,E2 -14762.463} C_VEL
LIN {X 0,Y 326.947,Z 359.384,A -85,B 0,C 180,E1 -14766.17,E2 -14766.17} C_VEL
LIN {X 0,Y 326.786,Z 359.398,A -85,B 0,C 180,E1 -14769.907,E2 -14769.907} C_VEL
LIN {X 0,Y 326.762,Z 359.404,A -85,B 0,C 180,E1 -14773.685,E2 -14773.685} C_VEL
LIN {X 0,Y 326.667,Z 359.418,A -85,B 0,C 180,E1 -14777.529,E2 -14777.529} C_VEL
LIN {X 0,Y 326.657,Z 359.42,A -85,B 0,C 180,E1 -14780.135,E2 -14780.135} C_VEL
LIN {X 0,Y 326.654,Z 359.415,A -85,B 0,C 180,E1 -14784.128,E2 -14784.128} C_VEL
LIN {X 0,Y 326.687,Z 359.413,A -85,B 0,C 180,E1 -14786.857,E2 -14786.857} C_VEL
LIN {X 0,Y 326.641,Z 359.42,A -85,B 0,C 180,E1 -14790.611,E2 -14790.611} C_VEL
LIN {X 0,Y 326.608,Z 359.427,A -85,B 0,C 180,E1 -14794.019,E2 -14794.019} C_VEL
LIN {X 0,Y 326.629,Z 359.423,A -85,B 0,C 180,E1 -14797.238,E2 -14797.238} C_VEL
LIN {X 0,Y 326.579,Z 359.429,A -85,B 0,C 180,E1 -14801.131,E2 -14801.131} C_VEL
LIN {X 0,Y 326.557,Z 359.432,A -85,B 0,C 180,E1 -14804.747,E2 -14804.747} C_VEL
LIN {X 0,Y 326.617,Z 359.608,A -85,B 0,C 180,E1 -14805.733,E2 -14805.733} C_VEL
LIN {X 0,Y 329.986,Z 369.502,A -85,B 0,C 180,E1 -14809.118,E2 -14809.118} C_VEL
LIN {X 0,Y 333.07,Z 379.931,A -85,B 0,C 180,E1 -14812.271,E2 -14812.271} C_VEL
LIN {X 0,Y 333.817,Z 382.512,A -85,B 0,C 180,E1 -14812.938,E2 -14812.938} C_VEL
LIN {X 0,Y 339.793,Z 393.998,A -85,B 0,C 180,E1 -14814.21,E2 -14814.21} C_VEL
LIN {X 0,Y 346.005,Z 407.125,A -85,B 0,C 180,E1 -14815.476,E2 -14815.476} C_VEL
LIN {X 0,Y 347.228,Z 410.466,A -85,B 0,C 180,E1 -14815.737,E2 -14815.737} C_VEL
LIN {X 0,Y 350.745,Z 432.649,A -85,B 0,C 180,E1 -14816.819,E2 -14816.819} C_VEL
LIN {X 0,Y 351.656,Z 440.037,A -85,B 0,C 180,E1 -14817.14,E2 -14817.14} C_VEL
LIN {X 0,Y 347.049,Z 551.904,A -85,B 0,C 180,E1 -14819.71,E2 -14819.71} C_VEL
LIN {X 0,Y 345.727,Z 567.92,A -85,B 0,C 180,E1 -14820.297,E2 -14820.297} C_VEL
LIN {X 0,Y 343.939,Z 582.699,A -85,B 0,C 180,E1 -14821.051,E2 -14821.051} C_VEL
LIN {X 0,Y 341.896,Z 597.148,A -85,B 0,C 180,E1 -14822.034,E2 -14822.034} C_VEL
LIN {X 0,Y 339.601,Z 611.155,A -85,B 0,C 180,E1 -14823.249,E2 -14823.249} C_VEL
LIN {X 0,Y 337.15,Z 624.622,A -85,B 0,C 180,E1 -14824.701,E2 -14824.701} C_VEL
LIN {X 0,Y 334.632,Z 636.969,A -85,B 0,C 180,E1 -14826.317,E2 -14826.317} C_VEL
LIN {X 0,Y 332.206,Z 649.483,A -85,B 0,C 180,E1 -14828.335,E2 -14828.335} C_VEL
LIN {X 0,Y 330.433,Z 658.659,A -85,B 0,C 180,E1 -14830.104,E2 -14830.104} C_VEL
LIN {X 0,Y 328.586,Z 668.005,A -85,B 0,C 180,E1 -14832.254,E2 -14832.254} C_VEL
LIN {X 0,Y 327.19,Z 675.808,A -85,B 0,C 180,E1 -14834.425,E2 -14834.425} C_VEL
LIN {X 0,Y 326.043,Z 683.145,A -85,B 0,C 180,E1 -14836.918,E2 -14836.918} C_VEL
LIN {X 0,Y 325.334,Z 688.977,A -85,B 0,C 180,E1 -14839.419,E2 -14839.419} C_VEL
LIN {X 0,Y 325.106,Z 692.488,A -85,B 0,C 180,E1 -14841.296,E2 -14841.296} C_VEL
LIN {X 0,Y 325.002,Z 695.974,A -85,B 0,C 180,E1 -14843.792,E2 -14843.792} C_VEL
LIN {X 0,Y 324.978,Z 698.205,A -85,B 0,C 180,E1 -14846.28,E2 -14846.28} C_VEL
LIN {X 0,Y 325.111,Z 699.248,A -85,B 0,C 180,E1 -14848.761,E2 -14848.761} C_VEL
LIN {X 0,Y 325.19,Z 699.326,A -85,B 0,C 180,E1 -14849.999,E2 -14849.999} C_VEL
LIN {X 0,Y 325.021,Z 698.564,A -85,B 0,C 180,E1 -14852.478,E2 -14852.478} C_VEL
LIN {X 0,Y 324.989,Z 696.592,A -85,B 0,C 180,E1 -14854.962,E2 -14854.962} C_VEL
LIN {X 0,Y 325.034,Z 693.323,A -85,B 0,C 180,E1 -14857.454,E2 -14857.454} C_VEL
LIN {X 0,Y 325.23,Z 688.714,A -85,B 0,C 180,E1 -14859.954,E2 -14859.954} C_VEL
LIN {X 0,Y 325.824,Z 682.671,A -85,B 0,C 180,E1 -14862.456,E2 -14862.456} C_VEL
LIN {X 0,Y 326.804,Z 675.03,A -85,B 0,C 180,E1 -14864.955,E2 -14864.955} C_VEL
LIN {X 0,Y 327.969,Z 666.818,A -85,B 0,C 180,E1 -14867.136,E2 -14867.136} C_VEL
LIN {X 0,Y 329.675,Z 656.96,A -85,B 0,C 180,E1 -14869.294,E2 -14869.294} C_VEL
LIN {X 0,Y 331.256,Z 646.849,A -85,B 0,C 180,E1 -14871.141,E2 -14871.141} C_VEL
LIN {X 0,Y 333.221,Z 634.836,A -85,B 0,C 180,E1 -14872.965,E2 -14872.965} C_VEL
LIN {X 0,Y 335.174,Z 622.879,A -85,B 0,C 180,E1 -14874.463,E2 -14874.463} C_VEL
LIN {X 0,Y 337.218,Z 609.987,A -85,B 0,C 180,E1 -14875.788,E2 -14875.788} C_VEL
LIN {X 0,Y 339.143,Z 596.053,A -85,B 0,C 180,E1 -14876.946,E2 -14876.946} C_VEL
LIN {X 0,Y 340.749,Z 581.504,A -85,B 0,C 180,E1 -14877.9,E2 -14877.9} C_VEL
LIN {X 0,Y 342.24,Z 565.985,A -85,B 0,C 180,E1 -14878.644,E2 -14878.644} C_VEL
LIN {X 0,Y 343.242,Z 550.9,A -85,B 0,C 180,E1 -14879.138,E2 -14879.138} C_VEL
LIN {X 0,Y 346.956,Z 439,A -85,B 0,C 180,E1 -14881.63,E2 -14881.63} C_VEL
LIN {X 0,Y 341.616,Z 406.035,A -85,B 0,C 180,E1 -14882.967,E2 -14882.967} C_VEL
LIN {X 0,Y 340.727,Z 402.528,A -85,B 0,C 180,E1 -14883.144,E2 -14883.144} C_VEL
LIN {X 0,Y 333.81,Z 386.242,A -85,B 0,C 180,E1 -14884.273,E2 -14884.273} C_VEL
LIN {X 0,Y 330.249,Z 372.49,A -85,B 0,C 180,E1 -14887.581,E2 -14887.581} C_VEL
LIN {X 0,Y 326.596,Z 359.435,A -85,B 0,C 180,E1 -14890.952,E2 -14890.952} C_VEL
LIN {X 0,Y 326.553,Z 359.432,A -85,B 0,C 180,E1 -14894.748,E2 -14894.748} C_VEL
LIN {X 0,Y 326.573,Z 359.425,A -85,B 0,C 180,E1 -14898.154,E2 -14898.154} C_VEL
LIN {X 0,Y 326.62,Z 359.423,A -85,B 0,C 180,E1 -14901.391,E2 -14901.391} C_VEL
LIN {X 0,Y 326.616,Z 359.427,A -85,B 0,C 180,E1 -14904.851,E2 -14904.851} C_VEL
LIN {X 0,Y 326.604,Z 359.427,A -85,B 0,C 180,E1 -14907.456,E2 -14907.456} C_VEL
LIN {X 0,Y 326.657,Z 359.419,A -85,B 0,C 180,E1 -14910.341,E2 -14910.341} C_VEL
LIN {X 0,Y 326.687,Z 359.414,A -85,B 0,C 180,E1 -14914.516,E2 -14914.516} C_VEL
LIN {X 0,Y 326.643,Z 359.42,A -85,B 0,C 180,E1 -14918.545,E2 -14918.545} C_VEL
LIN {X 0,Y 326.741,Z 359.41,A -85,B 0,C 180,E1 -14921.178,E2 -14921.178} C_VEL
LIN {X 0,Y 326.76,Z 359.406,A -85,B 0,C 180,E1 -14925.433,E2 -14925.433} C_VEL
LIN {X 0,Y 326.767,Z 359.399,A -85,B 0,C 180,E1 -14928.839,E2 -14928.839} C_VEL
LIN {X 0,Y 326.963,Z 359.379,A -85,B 0,C 180,E1 -14932.59,E2 -14932.59} C_VEL
LIN {X 0,Y 326.774,Z 359.407,A -85,B 0,C 180,E1 -14935.065,E2 -14935.065} C_VEL
LIN {X 0,Y 327.045,Z 359.365,A -85,B 0,C 180,E1 -14937.537,E2 -14937.537} C_VEL
LIN {X 0,Y 327.196,Z 359.347,A -85,B 0,C 180,E1 -14940,E2 -14940} C_VEL
LIN {X 0,Y 327.045,Z 359.371,A -85,B 0,C 180,E1 -14942.464,E2 -14942.464} C_VEL
LIN {X 0,Y 326.97,Z 359.373,A -85,B 0,C 180,E1 -14946.628,E2 -14946.628} C_VEL
LIN {X 0,Y 326.811,Z 359.397,A -85,B 0,C 180,E1 -14949.907,E2 -14949.907} C_VEL
LIN {X 0,Y 326.757,Z 359.403,A -85,B 0,C 180,E1 -14953.686,E2 -14953.686} C_VEL
LIN {X 0,Y 326.697,Z 359.409,A -85,B 0,C 180,E1 -14957.529,E2 -14957.529} C_VEL
LIN {X 0,Y 326.659,Z 359.417,A -85,B 0,C 180,E1 -14960.136,E2 -14960.136} C_VEL
LIN {X 0,Y 326.647,Z 359.417,A -85,B 0,C 180,E1 -14964.13,E2 -14964.13} C_VEL
LIN {X 0,Y 326.683,Z 359.415,A -85,B 0,C 180,E1 -14966.858,E2 -14966.858} C_VEL
LIN {X 0,Y 326.638,Z 359.425,A -85,B 0,C 180,E1 -14970.612,E2 -14970.612} C_VEL
LIN {X 0,Y 326.606,Z 359.421,A -85,B 0,C 180,E1 -14974.02,E2 -14974.02} C_VEL
LIN {X 0,Y 326.626,Z 359.421,A -85,B 0,C 180,E1 -14977.239,E2 -14977.239} C_VEL
LIN {X 0,Y 326.576,Z 359.427,A -85,B 0,C 180,E1 -14981.132,E2 -14981.132} C_VEL
LIN {X 0,Y 326.527,Z 359.436,A -85,B 0,C 180,E1 -14984.744,E2 -14984.744} C_VEL
LIN {X 0,Y 326.575,Z 359.43,A -85,B 0,C 180,E1 -14988.155,E2 -14988.155} C_VEL
LIN {X 0,Y 326.597,Z 359.42,A -85,B 0,C 180,E1 -14991.389,E2 -14991.389} C_VEL
LIN {X 0,Y 326.621,Z 359.425,A -85,B 0,C 180,E1 -14994.852,E2 -14994.852} C_VEL
LIN {X 0,Y 326.609,Z 359.421,A -85,B 0,C 180,E1 -14997.456,E2 -14997.456} C_VEL
LIN {X 0,Y 326.619,Z 359.425,A -85,B 0,C 180,E1 -15000.337,E2 -15000.337} C_VEL
LIN {X 0,Y 326.62,Z 359.421,A -85,B 0,C 180,E1 -15003.137,E2 -15003.137} C_VEL
LIN {X 0,Y 326.646,Z 359.419,A -85,B 0,C 180,E1 -15005.871,E2 -15005.871} C_VEL
LIN {X 0,Y 326.635,Z 359.422,A -85,B 0,C 180,E1 -15008.545,E2 -15008.545} C_VEL
LIN {X 0,Y 326.636,Z 359.424,A -85,B 0,C 180,E1 -15012.469,E2 -15012.469} C_VEL
LIN {X 0,Y 326.746,Z 359.412,A -85,B 0,C 180,E1 -15016.315,E2 -15016.315} C_VEL
LIN {X 0,Y 326.787,Z 359.405,A -85,B 0,C 180,E1 -15020.093,E2 -15020.093} C_VEL
LIN {X 0,Y 326.946,Z 359.384,A -85,B 0,C 180,E1 -15023.831,E2 -15023.831} C_VEL
LIN {X 0,Y 327.013,Z 359.373,A -85,B 0,C 180,E1 -15027.537,E2 -15027.537} C_VEL
LIN {X 0,Y 327.042,Z 359.37,A -85,B 0,C 180,E1 -15031.232,E2 -15031.232} C_VEL
LIN {X 0,Y 326.751,Z 359.404,A -85,B 0,C 180,E1 -15033.7,E2 -15033.7} C_VEL
LIN {X 0,Y 326.799,Z 359.402,A -85,B 0,C 180,E1 -15035.283,E2 -15035.283} C_VEL
LIN {X 0,Y 327.827,Z 362.182,A -85,B 0,C 180,E1 -15035.479,E2 -15035.479} C_VEL
LIN {X 0,Y 331.186,Z 368.066,A -85,B 0,C 180,E1 -15035.996,E2 -15035.996} C_VEL
LIN {X 0,Y 340.866,Z 386.719,A -85,B 0,C 180,E1 -15037.46,E2 -15037.46} C_VEL
LIN {X 0,Y 347.661,Z 400.741,A -85,B 0,C 180,E1 -15038.459,E2 -15038.459} C_VEL
LIN {X 0,Y 343.739,Z 517.404,A -85,B 0,C 180,E1 -15041.067,E2 -15041.067} C_VEL
LIN {X 0,Y 342.845,Z 532.574,A -85,B 0,C 180,E1 -15041.627,E2 -15041.627} C_VEL
LIN {X 0,Y 341.683,Z 547.208,A -85,B 0,C 180,E1 -15042.398,E2 -15042.398} C_VEL
LIN {X 0,Y 340.105,Z 562.208,A -85,B 0,C 180,E1 -15043.44,E2 -15043.44} C_VEL
LIN {X 0,Y 338.511,Z 575.172,A -85,B 0,C 180,E1 -15044.581,E2 -15044.581} C_VEL
LIN {X 0,Y 336.478,Z 589.161,A -85,B 0,C 180,E1 -15046.093,E2 -15046.093} C_VEL
LIN {X 0,Y 334.526,Z 601.508,A -85,B 0,C 180,E1 -15047.736,E2 -15047.736} C_VEL
LIN {X 0,Y 332.74,Z 612.133,A -85,B 0,C 180,E1 -15049.438,E2 -15049.438} C_VEL
LIN {X 0,Y 330.871,Z 622.848,A -85,B 0,C 180,E1 -15051.495,E2 -15051.495} C_VEL
LIN {X 0,Y 329.409,Z 631.264,A -85,B 0,C 180,E1 -15053.448,E2 -15053.448} C_VEL
LIN {X 0,Y 327.931,Z 639.768,A -85,B 0,C 180,E1 -15055.825,E2 -15055.825} C_VEL
LIN {X 0,Y 326.835,Z 646.69,A -85,B 0,C 180,E1 -15058.234,E2 -15058.234} C_VEL
LIN {X 0,Y 326.098,Z 651.759,A -85,B 0,C 180,E1 -15060.449,E2 -15060.449} C_VEL
LIN {X 0,Y 325.576,Z 655.75,A -85,B 0,C 180,E1 -15062.661,E2 -15062.661} C_VEL
LIN {X 0,Y 325.121,Z 658.591,A -85,B 0,C 180,E1 -15064.771,E2 -15064.771} C_VEL
LIN {X 0,Y 324.856,Z 660.828,A -85,B 0,C 180,E1 -15067.284,E2 -15067.284} C_VEL
LIN {X 0,Y 324.824,Z 661.547,A -85,B 0,C 180,E1 -15068.685,E2 -15068.685} C_VEL
LIN {X 0,Y 324.19,Z 661.975,A -85,B 0,C 180,E1 -15069.717,E2 -15069.717} C_VEL
LIN {X 0,Y 321.348,Z 662.225,A -85,B 0,C 180,E1 -15071.4,E2 -15071.4} C_VEL
LIN {X 0,Y 318.975,Z 661.997,A -85,B 0,C 180,E1 -15072.765,E2 -15072.765} C_VEL
LIN {X 0,Y 318.032,Z 661.622,A -85,B 0,C 180,E1 -15073.818,E2 -15073.818} C_VEL
LIN {X 0,Y 317.997,Z 661.38,A -85,B 0,C 180,E1 -15074.174,E2 -15074.174} C_VEL
LIN {X 0,Y 318.51,Z 659.324,A -85,B 0,C 180,E1 -15076.733,E2 -15076.733} C_VEL
LIN {X 0,Y 319.248,Z 655.676,A -85,B 0,C 180,E1 -15079.502,E2 -15079.502} C_VEL
LIN {X 0,Y 320.267,Z 650.685,A -85,B 0,C 180,E1 -15082.186,E2 -15082.186} C_VEL
LIN {X 0,Y 321.67,Z 644.417,A -85,B 0,C 180,E1 -15084.748,E2 -15084.748} C_VEL
LIN {X 0,Y 323.326,Z 637.239,A -85,B 0,C 180,E1 -15087.083,E2 -15087.083} C_VEL
LIN {X 0,Y 325.223,Z 629.081,A -85,B 0,C 180,E1 -15089.256,E2 -15089.256} C_VEL
LIN {X 0,Y 327.517,Z 619.555,A -85,B 0,C 180,E1 -15091.341,E2 -15091.341} C_VEL
LIN {X 0,Y 329.785,Z 609.126,A -85,B 0,C 180,E1 -15093.243,E2 -15093.243} C_VEL
LIN {X 0,Y 332.111,Z 597.758,A -85,B 0,C 180,E1 -15094.961,E2 -15094.961} C_VEL
LIN {X 0,Y 334.647,Z 584.578,A -85,B 0,C 180,E1 -15096.584,E2 -15096.584} C_VEL
LIN {X 0,Y 336.946,Z 570.881,A -85,B 0,C 180,E1 -15097.948,E2 -15097.948} C_VEL
LIN {X 0,Y 338.876,Z 556.559,A -85,B 0,C 180,E1 -15099.094,E2 -15099.094} C_VEL
LIN {X 0,Y 340.486,Z 541.437,A -85,B 0,C 180,E1 -15100.028,E2 -15100.028} C_VEL
LIN {X 0,Y 341.719,Z 526.191,A -85,B 0,C 180,E1 -15100.709,E2 -15100.709} C_VEL
LIN {X 0,Y 342.691,Z 508.851,A -85,B 0,C 180,E1 -15101.198,E2 -15101.198} C_VEL
LIN {X 0,Y 347.011,Z 406.568,A -85,B 0,C 180,E1 -15103.59,E2 -15103.59} C_VEL
LIN {X 0,Y 341.524,Z 395.514,A -85,B 0,C 180,E1 -15104.68,E2 -15104.68} C_VEL
LIN {X 0,Y 334.837,Z 384.07,A -85,B 0,C 180,E1 -15106.032,E2 -15106.032} C_VEL
LIN {X 0,Y 327.931,Z 373.182,A -85,B 0,C 180,E1 -15107.52,E2 -15107.52} C_VEL
LIN {X 0,Y 324.976,Z 368.919,A -85,B 0,C 180,E1 -15108.183,E2 -15108.183} C_VEL
LIN {X 0,Y 322.961,Z 365.716,A -85,B 0,C 180,E1 -15108.665,E2 -15108.665} C_VEL
LIN {X 0,Y 320.487,Z 362.716,A -85,B 0,C 180,E1 -15109.237,E2 -15109.237} C_VEL
LIN {X 0,Y 319.71,Z 360.289,A -85,B 0,C 180,E1 -15109.475,E2 -15109.475} C_VEL
LIN {X 0,Y 319.855,Z 360.267,A -85,B 0,C 180,E1 -15112.424,E2 -15112.424} C_VEL
LIN {X 0,Y 319.72,Z 360.281,A -85,B 0,C 180,E1 -15114.955,E2 -15114.955} C_VEL
LIN {X 0,Y 320.016,Z 360.248,A -85,B 0,C 180,E1 -15118.741,E2 -15118.741} C_VEL
LIN {X 0,Y 320.018,Z 360.246,A -85,B 0,C 180,E1 -15121.258,E2 -15121.258} C_VEL
LIN {X 0,Y 319.732,Z 360.28,A -85,B 0,C 180,E1 -15123.781,E2 -15123.781} C_VEL
LIN {X 0,Y 319.904,Z 360.261,A -85,B 0,C 180,E1 -15126.306,E2 -15126.306} C_VEL
LIN {X 0,Y 319.738,Z 360.276,A -85,B 0,C 180,E1 -15130.127,E2 -15130.127} C_VEL
LIN {X 0,Y 319.735,Z 360.282,A -85,B 0,C 180,E1 -15133.992,E2 -15133.992} C_VEL
LIN {X 0,Y 319.627,Z 360.292,A -85,B 0,C 180,E1 -15137.928,E2 -15137.928} C_VEL
LIN {X 0,Y 319.611,Z 360.297,A -85,B 0,C 180,E1 -15140.599,E2 -15140.599} C_VEL
LIN {X 0,Y 319.572,Z 360.302,A -85,B 0,C 180,E1 -15143.319,E2 -15143.319} C_VEL
LIN {X 0,Y 319.637,Z 360.295,A -85,B 0,C 180,E1 -15146.087,E2 -15146.087} C_VEL
LIN {X 0,Y 319.592,Z 360.3,A -85,B 0,C 180,E1 -15148.933,E2 -15148.933} C_VEL
LIN {X 0,Y 319.534,Z 360.305,A -85,B 0,C 180,E1 -15151.861,E2 -15151.861} C_VEL
LIN {X 0,Y 319.581,Z 360.303,A -85,B 0,C 180,E1 -15155.542,E2 -15155.542} C_VEL
LIN {X 0,Y 319.574,Z 360.306,A -85,B 0,C 180,E1 -15158.007,E2 -15158.007} C_VEL
LIN {X 0,Y 319.527,Z 360.308,A -85,B 0,C 180,E1 -15161.596,E2 -15161.596} C_VEL
LIN {X 0,Y 319.535,Z 360.401,A -85,B 0,C 180,E1 -15164.517,E2 -15164.517} C_VEL
LIN {X 0,Y 322.606,Z 369.335,A -85,B 0,C 180,E1 -15167.79,E2 -15167.79} C_VEL
LIN {X 0,Y 325.687,Z 379.152,A -85,B 0,C 180,E1 -15170.972,E2 -15170.972} C_VEL
LIN {X 0,Y 326.488,Z 381.801,A -85,B 0,C 180,E1 -15171.709,E2 -15171.709} C_VEL
LIN {X 0,Y 333.582,Z 395.134,A -85,B 0,C 180,E1 -15173.312,E2 -15173.312} C_VEL
LIN {X 0,Y 340.006,Z 408.534,A -85,B 0,C 180,E1 -15174.687,E2 -15174.687} C_VEL
LIN {X 0,Y 342.011,Z 413.666,A -85,B 0,C 180,E1 -15175.125,E2 -15175.125} C_VEL
LIN {X 0,Y 345.199,Z 434.922,A -85,B 0,C 180,E1 -15176.184,E2 -15176.184} C_VEL
LIN {X 0,Y 345.946,Z 441.489,A -85,B 0,C 180,E1 -15176.47,E2 -15176.47} C_VEL
LIN {X 0,Y 341.173,Z 551.514,A -85,B 0,C 180,E1 -15179.046,E2 -15179.046} C_VEL
LIN {X 0,Y 339.748,Z 567.437,A -85,B 0,C 180,E1 -15179.634,E2 -15179.634} C_VEL
LIN {X 0,Y 337.778,Z 583.307,A -85,B 0,C 180,E1 -15180.471,E2 -15180.471} C_VEL
LIN {X 0,Y 335.621,Z 597.709,A -85,B 0,C 180,E1 -15181.481,E2 -15181.481} C_VEL
LIN {X 0,Y 333.289,Z 611.383,A -85,B 0,C 180,E1 -15182.7,E2 -15182.7} C_VEL
LIN {X 0,Y 330.744,Z 624.736,A -85,B 0,C 180,E1 -15184.176,E2 -15184.176} C_VEL
LIN {X 0,Y 328.372,Z 635.981,A -85,B 0,C 180,E1 -15185.669,E2 -15185.669} C_VEL
LIN {X 0,Y 325.974,Z 647.368,A -85,B 0,C 180,E1 -15187.499,E2 -15187.499} C_VEL
LIN {X 0,Y 323.708,Z 658.512,A -85,B 0,C 180,E1 -15189.673,E2 -15189.673} C_VEL
LIN {X 0,Y 321.744,Z 667.822,A -85,B 0,C 180,E1 -15191.864,E2 -15191.864} C_VEL
LIN {X 0,Y 320.277,Z 675.586,A -85,B 0,C 180,E1 -15194.08,E2 -15194.08} C_VEL
LIN {X 0,Y 319.056,Z 682.883,A -85,B 0,C 180,E1 -15196.626,E2 -15196.626} C_VEL
LIN {X 0,Y 318.294,Z 688.67,A -85,B 0,C 180,E1 -15199.182,E2 -15199.182} C_VEL
LIN {X 0,Y 318.039,Z 692.144,A -85,B 0,C 180,E1 -15201.101,E2 -15201.101} C_VEL
LIN {X 0,Y 317.902,Z 695.62,A -85,B 0,C 180,E1 -15203.653,E2 -15203.653} C_VEL
LIN {X 0,Y 317.903,Z 697.827,A -85,B 0,C 180,E1 -15206.197,E2 -15206.197} C_VEL
LIN {X 0,Y 318.016,Z 698.841,A -85,B 0,C 180,E1 -15208.733,E2 -15208.733} C_VEL
LIN {X 0,Y 318.114,Z 698.905,A -85,B 0,C 180,E1 -15209.999,E2 -15209.999} C_VEL
LIN {X 0,Y 317.93,Z 698.111,A -85,B 0,C 180,E1 -15212.533,E2 -15212.533} C_VEL
LIN {X 0,Y 317.897,Z 696.109,A -85,B 0,C 180,E1 -15215.073,E2 -15215.073} C_VEL
LIN {X 0,Y 317.959,Z 692.818,A -85,B 0,C 180,E1 -15217.62,E2 -15217.62} C_VEL
LIN {X 0,Y 318.179,Z 688.169,A -85,B 0,C 180,E1 -15220.177,E2 -15220.177} C_VEL
LIN {X 0,Y 318.795,Z 682.08,A -85,B 0,C 180,E1 -15222.735,E2 -15222.735} C_VEL
LIN {X 0,Y 319.842,Z 674.392,A -85,B 0,C 180,E1 -15225.288,E2 -15225.288} C_VEL
LIN {X 0,Y 321.091,Z 666.126,A -85,B 0,C 180,E1 -15227.515,E2 -15227.515} C_VEL
LIN {X 0,Y 322.87,Z 656.206,A -85,B 0,C 180,E1 -15229.717,E2 -15229.717} C_VEL
LIN {X 0,Y 324.529,Z 646.021,A -85,B 0,C 180,E1 -15231.601,E2 -15231.601} C_VEL
LIN {X 0,Y 326.415,Z 635.013,A -85,B 0,C 180,E1 -15233.305,E2 -15233.305} C_VEL
LIN {X 0,Y 328.425,Z 623.171,A -85,B 0,C 180,E1 -15234.831,E2 -15234.831} C_VEL
LIN {X 0,Y 330.535,Z 610.432,A -85,B 0,C 180,E1 -15236.18,E2 -15236.18} C_VEL
LIN {X 0,Y 332.521,Z 596.545,A -85,B 0,C 180,E1 -15237.371,E2 -15237.371} C_VEL
LIN {X 0,Y 334.152,Z 582.469,A -85,B 0,C 180,E1 -15238.329,E2 -15238.329} C_VEL
LIN {X 0,Y 335.7,Z 567.495,A -85,B 0,C 180,E1 -15239.083,E2 -15239.083} C_VEL
LIN {X 0,Y 336.802,Z 552.129,A -85,B 0,C 180,E1 -15239.622,E2 -15239.622} C_VEL
LIN {X 0,Y 340.688,Z 440.13,A -85,B 0,C 180,E1 -15242.169,E2 -15242.169} C_VEL
LIN {X 0,Y 336.016,Z 410.658,A -85,B 0,C 180,E1 -15243.38,E2 -15243.38} C_VEL
LIN {X 0,Y 334.749,Z 405.021,A -85,B 0,C 180,E1 -15243.654,E2 -15243.654} C_VEL
LIN {X 0,Y 326.449,Z 385.844,A -85,B 0,C 180,E1 -15245.037,E2 -15245.037} C_VEL
LIN {X 0,Y 323.232,Z 373.558,A -85,B 0,C 180,E1 -15248.078,E2 -15248.078} C_VEL
LIN {X 0,Y 320.427,Z 363.445,A -85,B 0,C 180,E1 -15250.722,E2 -15250.722} C_VEL
LIN {X 0,Y 319.523,Z 360.309,A -85,B 0,C 180,E1 -15251.597,E2 -15251.597} C_VEL
LIN {X 0,Y 319.512,Z 360.309,A -85,B 0,C 180,E1 -15254.738,E2 -15254.738} C_VEL
LIN {X 0,Y 319.557,Z 360.306,A -85,B 0,C 180,E1 -15257.018,E2 -15257.018} C_VEL
LIN {X 0,Y 319.543,Z 360.305,A -85,B 0,C 180,E1 -15260.371,E2 -15260.371} C_VEL
LIN {X 0,Y 319.555,Z 360.307,A -85,B 0,C 180,E1 -15263.572,E2 -15263.572} C_VEL
LIN {X 0,Y 319.573,Z 360.299,A -85,B 0,C 180,E1 -15266.686,E2 -15266.686} C_VEL
LIN {X 0,Y 319.587,Z 360.301,A -85,B 0,C 180,E1 -15269.617,E2 -15269.617} C_VEL
LIN {X 0,Y 319.605,Z 360.298,A -85,B 0,C 180,E1 -15272.498,E2 -15272.498} C_VEL
LIN {X 0,Y 319.602,Z 360.3,A -85,B 0,C 180,E1 -15275.304,E2 -15275.304} C_VEL
LIN {X 0,Y 319.593,Z 360.296,A -85,B 0,C 180,E1 -15278.048,E2 -15278.048} C_VEL
LIN {X 0,Y 319.685,Z 360.29,A -85,B 0,C 180,E1 -15280.963,E2 -15280.963} C_VEL
LIN {X 0,Y 319.728,Z 360.283,A -85,B 0,C 180,E1 -15285.276,E2 -15285.276} C_VEL
LIN {X 0,Y 319.754,Z 360.268,A -85,B 0,C 180,E1 -15289.873,E2 -15289.873} C_VEL
LIN {X 0,Y 319.922,Z 360.255,A -85,B 0,C 180,E1 -15292.426,E2 -15292.426} C_VEL
LIN {X 0,Y 319.743,Z 360.283,A -85,B 0,C 180,E1 -15294.956,E2 -15294.956} C_VEL
LIN {X 0,Y 319.989,Z 360.244,A -85,B 0,C 180,E1 -15297.483,E2 -15297.483} C_VEL
LIN {X 0,Y 320.148,Z 360.225,A -85,B 0,C 180,E1 -15300,E2 -15300} C_VEL
LIN {X 0,Y 319.989,Z 360.25,A -85,B 0,C 180,E1 -15302.518,E2 -15302.518} C_VEL
LIN {X 0,Y 319.931,Z 360.25,A -85,B 0,C 180,E1 -15306.618,E2 -15306.618} C_VEL
LIN {X 0,Y 319.756,Z 360.276,A -85,B 0,C 180,E1 -15310.128,E2 -15310.128} C_VEL
LIN {X 0,Y 319.729,Z 360.281,A -85,B 0,C 180,E1 -15314.725,E2 -15314.725} C_VEL
LIN {X 0,Y 319.687,Z 360.288,A -85,B 0,C 180,E1 -15319.038,E2 -15319.038} C_VEL
LIN {X 0,Y 319.558,Z 360.3,A -85,B 0,C 180,E1 -15323.321,E2 -15323.321} C_VEL
LIN {X 0,Y 319.617,Z 360.287,A -85,B 0,C 180,E1 -15326.09,E2 -15326.09} C_VEL
LIN {X 0,Y 319.589,Z 360.301,A -85,B 0,C 180,E1 -15328.934,E2 -15328.934} C_VEL
LIN {X 0,Y 319.531,Z 360.305,A -85,B 0,C 180,E1 -15331.863,E2 -15331.863} C_VEL
LIN {X 0,Y 319.579,Z 360.293,A -85,B 0,C 180,E1 -15335.544,E2 -15335.544} C_VEL
LIN {X 0,Y 319.556,Z 360.302,A -85,B 0,C 180,E1 -15338.011,E2 -15338.011} C_VEL
LIN {X 0,Y 319.525,Z 360.304,A -85,B 0,C 180,E1 -15341.598,E2 -15341.598} C_VEL
LIN {X 0,Y 319.488,Z 360.31,A -85,B 0,C 180,E1 -15345.258,E2 -15345.258} C_VEL
LIN {X 0,Y 319.528,Z 360.308,A -85,B 0,C 180,E1 -15348.712,E2 -15348.712} C_VEL
LIN {X 0,Y 319.554,Z 360.301,A -85,B 0,C 180,E1 -15352.351,E2 -15352.351} C_VEL
LIN {X 0,Y 319.561,Z 360.302,A -85,B 0,C 180,E1 -15355.124,E2 -15355.124} C_VEL
LIN {X 0,Y 319.525,Z 360.305,A -85,B 0,C 180,E1 -15358.138,E2 -15358.138} C_VEL
LIN {X 0,Y 319.59,Z 360.298,A -85,B 0,C 180,E1 -15361.599,E2 -15361.599} C_VEL
LIN {X 0,Y 319.584,Z 360.297,A -85,B 0,C 180,E1 -15365.303,E2 -15365.303} C_VEL
LIN {X 0,Y 319.591,Z 360.3,A -85,B 0,C 180,E1 -15368.048,E2 -15368.048} C_VEL
LIN {X 0,Y 319.59,Z 360.301,A -85,B 0,C 180,E1 -15372.07,E2 -15372.07} C_VEL
LIN {X 0,Y 319.712,Z 360.285,A -85,B 0,C 180,E1 -15376.008,E2 -15376.008} C_VEL
LIN {X 0,Y 319.739,Z 360.281,A -85,B 0,C 180,E1 -15379.873,E2 -15379.873} C_VEL
LIN {X 0,Y 319.903,Z 360.261,A -85,B 0,C 180,E1 -15383.694,E2 -15383.694} C_VEL
LIN {X 0,Y 319.959,Z 360.252,A -85,B 0,C 180,E1 -15387.483,E2 -15387.483} C_VEL
LIN {X 0,Y 320.011,Z 360.247,A -85,B 0,C 180,E1 -15391.259,E2 -15391.259} C_VEL
LIN {X 0,Y 319.715,Z 360.287,A -85,B 0,C 180,E1 -15394.532,E2 -15394.532} C_VEL
LIN {X 0,Y 320.75,Z 363.17,A -85,B 0,C 180,E1 -15394.736,E2 -15394.736} C_VEL
LIN {X 0,Y 322.539,Z 366.181,A -85,B 0,C 180,E1 -15395.02,E2 -15395.02} C_VEL
LIN {X 0,Y 328.004,Z 375.936,A -85,B 0,C 180,E1 -15395.88,E2 -15395.88} C_VEL
LIN {X 0,Y 341.026,Z 401.995,A -85,B 0,C 180,E1 -15397.875,E2 -15397.875} C_VEL
LIN {X 0,Y 341.346,Z 402.664,A -85,B 0,C 180,E1 -15397.922,E2 -15397.922} C_VEL
LIN {X 0,Y 337.374,Z 517.602,A -85,B 0,C 180,E1 -15400.541,E2 -15400.541} C_VEL
LIN {X 0,Y 336.429,Z 533.088,A -85,B 0,C 180,E1 -15401.123,E2 -15401.123} C_VEL
LIN {X 0,Y 335.177,Z 548.246,A -85,B 0,C 180,E1 -15401.942,E2 -15401.942} C_VEL
LIN {X 0,Y 333.634,Z 562.279,A -85,B 0,C 180,E1 -15402.934,E2 -15402.934} C_VEL
LIN {X 0,Y 331.815,Z 576.648,A -85,B 0,C 180,E1 -15404.228,E2 -15404.228} C_VEL
LIN {X 0,Y 329.935,Z 589.068,A -85,B 0,C 180,E1 -15405.601,E2 -15405.601} C_VEL
LIN {X 0,Y 327.886,Z 601.586,A -85,B 0,C 180,E1 -15407.286,E2 -15407.286} C_VEL
LIN {X 0,Y 325.848,Z 613.305,A -85,B 0,C 180,E1 -15409.204,E2 -15409.204} C_VEL
LIN {X 0,Y 323.882,Z 624.091,A -85,B 0,C 180,E1 -15411.35,E2 -15411.35} C_VEL
LIN {X 0,Y 322.198,Z 633.485,A -85,B 0,C 180,E1 -15413.632,E2 -15413.632} C_VEL
LIN {X 0,Y 320.741,Z 641.617,A -85,B 0,C 180,E1 -15416.053,E2 -15416.053} C_VEL
LIN {X 0,Y 319.666,Z 648.068,A -85,B 0,C 180,E1 -15418.427,E2 -15418.427} C_VEL
LIN {X 0,Y 318.956,Z 653.065,A -85,B 0,C 180,E1 -15420.756,E2 -15420.756} C_VEL
LIN {X 0,Y 318.284,Z 657.522,A -85,B 0,C 180,E1 -15423.506,E2 -15423.506} C_VEL
LIN {X 0,Y 317.998,Z 659.475,A -85,B 0,C 180,E1 -15425.141,E2 -15425.141} C_VEL
LIN {X 0,Y 317.777,Z 661.204,A -85,B 0,C 180,E1 -15427.232,E2 -15427.232} C_VEL
LIN {X 0,Y 317.731,Z 662.302,A -85,B 0,C 180,E1 -15429.902,E2 -15429.902} C_VEL
LIN {X 0,Y 317.761,Z 662.349,A -85,B 0,C 180,E1 -15431.569,E2 -15431.569} C_VEL
LIN {X 0,Y 317.997,Z 661.38,A -85,B 0,C 180,E1 -15434.174,E2 -15434.174} C_VEL
LIN {X 0,Y 317.503,Z 660.772,A -85,B 0,C 180,E1 -15435.229,E2 -15435.229} C_VEL
LIN {X 0,Y 314.992,Z 659.46,A -85,B 0,C 180,E1 -15436.953,E2 -15436.953} C_VEL
LIN {X 0,Y 312.929,Z 658.07,A -85,B 0,C 180,E1 -15438.337,E2 -15438.337} C_VEL
LIN {X 0,Y 312.211,Z 656.73,A -85,B 0,C 180,E1 -15439.388,E2 -15439.388} C_VEL
LIN {X 0,Y 312.245,Z 656.181,A -85,B 0,C 180,E1 -15439.738,E2 -15439.738} C_VEL
LIN {X 0,Y 313.023,Z 652.616,A -85,B 0,C 180,E1 -15441.797,E2 -15441.797} C_VEL
LIN {X 0,Y 314.42,Z 646.652,A -85,B 0,C 180,E1 -15444.467,E2 -15444.467} C_VEL
LIN {X 0,Y 316.115,Z 639.734,A -85,B 0,C 180,E1 -15446.903,E2 -15446.903} C_VEL
LIN {X 0,Y 317.999,Z 632.141,A -85,B 0,C 180,E1 -15449.08,E2 -15449.08} C_VEL
LIN {X 0,Y 320.384,Z 622.563,A -85,B 0,C 180,E1 -15451.337,E2 -15451.337} C_VEL
LIN {X 0,Y 322.88,Z 611.981,A -85,B 0,C 180,E1 -15453.384,E2 -15453.384} C_VEL
LIN {X 0,Y 325.284,Z 600.929,A -85,B 0,C 180,E1 -15455.155,E2 -15455.155} C_VEL
LIN {X 0,Y 327.905,Z 588.074,A -85,B 0,C 180,E1 -15456.851,E2 -15456.851} C_VEL
LIN {X 0,Y 330.42,Z 574.352,A -85,B 0,C 180,E1 -15458.311,E2 -15458.311} C_VEL
LIN {X 0,Y 332.313,Z 561.606,A -85,B 0,C 180,E1 -15459.414,E2 -15459.414} C_VEL
LIN {X 0,Y 334.146,Z 546.963,A -85,B 0,C 180,E1 -15460.411,E2 -15460.411} C_VEL
LIN {X 0,Y 335.538,Z 532.044,A -85,B 0,C 180,E1 -15461.174,E2 -15461.174} C_VEL
LIN {X 0,Y 336.523,Z 517.558,A -85,B 0,C 180,E1 -15461.683,E2 -15461.683} C_VEL
LIN {X 0,Y 341.46,Z 409.004,A -85,B 0,C 180,E1 -15464.277,E2 -15464.277} C_VEL
LIN {X 0,Y 335.74,Z 397.767,A -85,B 0,C 180,E1 -15465.451,E2 -15465.451} C_VEL
LIN {X 0,Y 327.897,Z 384.544,A -85,B 0,C 180,E1 -15467.134,E2 -15467.134} C_VEL
LIN {X 0,Y 322.92,Z 376.826,A -85,B 0,C 180,E1 -15468.271,E2 -15468.271} C_VEL
LIN {X 0,Y 320.74,Z 373.688,A -85,B 0,C 180,E1 -15468.786,E2 -15468.786} C_VEL
LIN {X 0,Y 318.427,Z 370.267,A -85,B 0,C 180,E1 -15469.347,E2 -15469.347} C_VEL
LIN {X 0,Y 316.283,Z 367.194,A -85,B 0,C 180,E1 -15469.881,E2 -15469.881} C_VEL
LIN {X 0,Y 315.61,Z 366.033,A -85,B 0,C 180,E1 -15470.062,E2 -15470.062} C_VEL
LIN {X 0,Y 313.679,Z 363.889,A -85,B 0,C 180,E1 -15470.542,E2 -15470.542} C_VEL
LIN {X 0,Y 312.758,Z 361.15,A -85,B 0,C 180,E1 -15470.868,E2 -15470.868} C_VEL
LIN {X 0,Y 312.842,Z 361.141,A -85,B 0,C 180,E1 -15473.55,E2 -15473.55} C_VEL
LIN {X 0,Y 312.983,Z 361.124,A -85,B 0,C 180,E1 -15478.713,E2 -15478.713} C_VEL
LIN {X 0,Y 312.986,Z 361.121,A -85,B 0,C 180,E1 -15481.286,E2 -15481.286} C_VEL
LIN {X 0,Y 312.682,Z 361.158,A -85,B 0,C 180,E1 -15483.866,E2 -15483.866} C_VEL
LIN {X 0,Y 312.845,Z 361.14,A -85,B 0,C 180,E1 -15486.449,E2 -15486.449} C_VEL
LIN {X 0,Y 312.753,Z 361.152,A -85,B 0,C 180,E1 -15489.05,E2 -15489.05} C_VEL
LIN {X 0,Y 312.637,Z 361.16,A -85,B 0,C 180,E1 -15492.991,E2 -15492.991} C_VEL
LIN {X 0,Y 312.624,Z 361.161,A -85,B 0,C 180,E1 -15495.65,E2 -15495.65} C_VEL
LIN {X 0,Y 312.58,Z 361.172,A -85,B 0,C 180,E1 -15499.709,E2 -15499.709} C_VEL
LIN {X 0,Y 312.548,Z 361.177,A -85,B 0,C 180,E1 -15502.789,E2 -15502.789} C_VEL
LIN {X 0,Y 312.605,Z 361.171,A -85,B 0,C 180,E1 -15505.935,E2 -15505.935} C_VEL
LIN {X 0,Y 312.547,Z 361.173,A -85,B 0,C 180,E1 -15509.649,E2 -15509.649} C_VEL
LIN {X 0,Y 312.521,Z 361.183,A -85,B 0,C 180,E1 -15513.688,E2 -15513.688} C_VEL
LIN {X 0,Y 312.538,Z 361.178,A -85,B 0,C 180,E1 -15517.383,E2 -15517.383} C_VEL
LIN {X 0,Y 312.491,Z 361.186,A -85,B 0,C 180,E1 -15520.709,E2 -15520.709} C_VEL
LIN {X 0,Y 312.527,Z 361.186,A -85,B 0,C 180,E1 -15523.193,E2 -15523.193} C_VEL
LIN {X 0,Y 315.587,Z 370.311,A -85,B 0,C 180,E1 -15526.736,E2 -15526.736} C_VEL
LIN {X 0,Y 318.474,Z 379.175,A -85,B 0,C 180,E1 -15529.803,E2 -15529.803} C_VEL
LIN {X 0,Y 319.054,Z 380.978,A -85,B 0,C 180,E1 -15530.345,E2 -15530.345} C_VEL
LIN {X 0,Y 325.697,Z 393.007,A -85,B 0,C 180,E1 -15531.962,E2 -15531.962} C_VEL
LIN {X 0,Y 330.377,Z 402.128,A -85,B 0,C 180,E1 -15533.039,E2 -15533.039} C_VEL
LIN {X 0,Y 336.665,Z 415.967,A -85,B 0,C 180,E1 -15534.439,E2 -15534.439} C_VEL
LIN {X 0,Y 339.687,Z 436.739,A -85,B 0,C 180,E1 -15535.502,E2 -15535.502} C_VEL
LIN {X 0,Y 340.325,Z 442.239,A -85,B 0,C 180,E1 -15535.756,E2 -15535.756} C_VEL
LIN {X 0,Y 335.44,Z 550.321,A -85,B 0,C 180,E1 -15538.325,E2 -15538.325} C_VEL
LIN {X 0,Y 333.958,Z 566.482,A -85,B 0,C 180,E1 -15538.918,E2 -15538.918} C_VEL
LIN {X 0,Y 332.011,Z 581.872,A -85,B 0,C 180,E1 -15539.73,E2 -15539.73} C_VEL
LIN {X 0,Y 329.637,Z 596.847,A -85,B 0,C 180,E1 -15540.781,E2 -15540.781} C_VEL
LIN {X 0,Y 327.285,Z 610.211,A -85,B 0,C 180,E1 -15541.982,E2 -15541.982} C_VEL
LIN {X 0,Y 324.616,Z 623.67,A -85,B 0,C 180,E1 -15543.478,E2 -15543.478} C_VEL
LIN {X 0,Y 321.897,Z 636.023,A -85,B 0,C 180,E1 -15545.147,E2 -15545.147} C_VEL
LIN {X 0,Y 319.393,Z 647.352,A -85,B 0,C 180,E1 -15547.009,E2 -15547.009} C_VEL
LIN {X 0,Y 316.995,Z 658.406,A -85,B 0,C 180,E1 -15549.222,E2 -15549.222} C_VEL
LIN {X 0,Y 314.916,Z 667.649,A -85,B 0,C 180,E1 -15551.456,E2 -15551.456} C_VEL
LIN {X 0,Y 313.36,Z 675.364,A -85,B 0,C 180,E1 -15553.718,E2 -15553.718} C_VEL
LIN {X 0,Y 312.079,Z 682.626,A -85,B 0,C 180,E1 -15556.322,E2 -15556.322} C_VEL
LIN {X 0,Y 311.27,Z 688.378,A -85,B 0,C 180,E1 -15558.935,E2 -15558.935} C_VEL
LIN {X 0,Y 310.96,Z 691.817,A -85,B 0,C 180,E1 -15560.897,E2 -15560.897} C_VEL
LIN {X 0,Y 310.817,Z 695.272,A -85,B 0,C 180,E1 -15563.508,E2 -15563.508} C_VEL
LIN {X 0,Y 310.828,Z 697.45,A -85,B 0,C 180,E1 -15566.11,E2 -15566.11} C_VEL
LIN {X 0,Y 310.921,Z 698.435,A -85,B 0,C 180,E1 -15568.704,E2 -15568.704} C_VEL
LIN {X 0,Y 311.024,Z 698.484,A -85,B 0,C 180,E1 -15569.999,E2 -15569.999} C_VEL
LIN {X 0,Y 310.843,Z 697.659,A -85,B 0,C 180,E1 -15572.591,E2 -15572.591} C_VEL
LIN {X 0,Y 310.81,Z 695.623,A -85,B 0,C 180,E1 -15575.189,E2 -15575.189} C_VEL
LIN {X 0,Y 310.882,Z 692.31,A -85,B 0,C 180,E1 -15577.795,E2 -15577.795} C_VEL
LIN {X 0,Y 311.112,Z 687.623,A -85,B 0,C 180,E1 -15580.411,E2 -15580.411} C_VEL
LIN {X 0,Y 311.781,Z 681.49,A -85,B 0,C 180,E1 -15583.027,E2 -15583.027} C_VEL
LIN {X 0,Y 312.904,Z 673.755,A -85,B 0,C 180,E1 -15585.635,E2 -15585.635} C_VEL
LIN {X 0,Y 314.213,Z 665.434,A -85,B 0,C 180,E1 -15587.911,E2 -15587.911} C_VEL
LIN {X 0,Y 315.82,Z 656.972,A -85,B 0,C 180,E1 -15589.837,E2 -15589.837} C_VEL
LIN {X 0,Y 317.617,Z 646.354,A -85,B 0,C 180,E1 -15591.875,E2 -15591.875} C_VEL
LIN {X 0,Y 319.619,Z 635.162,A -85,B 0,C 180,E1 -15593.658,E2 -15593.658} C_VEL
LIN {X 0,Y 321.686,Z 623.417,A -85,B 0,C 180,E1 -15595.215,E2 -15595.215} C_VEL
LIN {X 0,Y 323.848,Z 610.806,A -85,B 0,C 180,E1 -15596.589,E2 -15596.589} C_VEL
LIN {X 0,Y 325.917,Z 597.042,A -85,B 0,C 180,E1 -15597.804,E2 -15597.804} C_VEL
LIN {X 0,Y 327.719,Z 582.007,A -85,B 0,C 180,E1 -15598.849,E2 -15598.849} C_VEL
LIN {X 0,Y 329.288,Z 567.001,A -85,B 0,C 180,E1 -15599.618,E2 -15599.618} C_VEL
LIN {X 0,Y 330.417,Z 551.591,A -85,B 0,C 180,E1 -15600.165,E2 -15600.165} C_VEL
LIN {X 0,Y 334.424,Z 441.688,A -85,B 0,C 180,E1 -15602.706,E2 -15602.706} C_VEL
LIN {X 0,Y 330.704,Z 417.153,A -85,B 0,C 180,E1 -15603.723,E2 -15603.723} C_VEL
LIN {X 0,Y 329.082,Z 408.298,A -85,B 0,C 180,E1 -15604.127,E2 -15604.127} C_VEL
LIN {X 0,Y 320.476,Z 388.614,A -85,B 0,C 180,E1 -15605.586,E2 -15605.586} C_VEL
LIN {X 0,Y 319.085,Z 385.303,A -85,B 0,C 180,E1 -15605.866,E2 -15605.866} C_VEL
LIN {X 0,Y 315.549,Z 371.968,A -85,B 0,C 180,E1 -15609.29,E2 -15609.29} C_VEL
LIN {X 0,Y 312.482,Z 361.185,A -85,B 0,C 180,E1 -15612.26,E2 -15612.26} C_VEL
LIN {X 0,Y 312.478,Z 361.187,A -85,B 0,C 180,E1 -15616.03,E2 -15616.03} C_VEL
LIN {X 0,Y 312.5,Z 361.183,A -85,B 0,C 180,E1 -15619.874,E2 -15619.874} C_VEL
LIN {X 0,Y 312.532,Z 361.18,A -85,B 0,C 180,E1 -15624.05,E2 -15624.05} C_VEL
LIN {X 0,Y 312.501,Z 361.182,A -85,B 0,C 180,E1 -15627.334,E2 -15627.334} C_VEL
LIN {X 0,Y 312.549,Z 361.179,A -85,B 0,C 180,E1 -15631.276,E2 -15631.276} C_VEL
LIN {X 0,Y 312.582,Z 361.172,A -85,B 0,C 180,E1 -15634.711,E2 -15634.711} C_VEL
LIN {X 0,Y 312.584,Z 361.171,A -85,B 0,C 180,E1 -15637.529,E2 -15637.529} C_VEL
LIN {X 0,Y 312.635,Z 361.163,A -85,B 0,C 180,E1 -15641.657,E2 -15641.657} C_VEL
LIN {X 0,Y 312.69,Z 361.157,A -85,B 0,C 180,E1 -15645.686,E2 -15645.686} C_VEL
LIN {X 0,Y 312.698,Z 361.147,A -85,B 0,C 180,E1 -15649.642,E2 -15649.642} C_VEL
LIN {X 0,Y 312.863,Z 361.133,A -85,B 0,C 180,E1 -15652.254,E2 -15652.254} C_VEL
LIN {X 0,Y 312.713,Z 361.159,A -85,B 0,C 180,E1 -15654.843,E2 -15654.843} C_VEL
LIN {X 0,Y 312.988,Z 361.117,A -85,B 0,C 180,E1 -15658.714,E2 -15658.714} C_VEL
LIN {X 0,Y 312.988,Z 361.122,A -85,B 0,C 180,E1 -15661.287,E2 -15661.287} C_VEL
LIN {X 0,Y 312.716,Z 361.152,A -85,B 0,C 180,E1 -15665.158,E2 -15665.158} C_VEL
LIN {X 0,Y 312.87,Z 361.128,A -85,B 0,C 180,E1 -15667.746,E2 -15667.746} C_VEL
LIN {X 0,Y 312.667,Z 361.16,A -85,B 0,C 180,E1 -15671.672,E2 -15671.672} C_VEL
LIN {X 0,Y 312.698,Z 361.154,A -85,B 0,C 180,E1 -15674.888,E2 -15674.888} C_VEL
LIN {X 0,Y 312.628,Z 361.166,A -85,B 0,C 180,E1 -15679.237,E2 -15679.237} C_VEL
LIN {X 0,Y 312.524,Z 361.18,A -85,B 0,C 180,E1 -15682.781,E2 -15682.781} C_VEL
LIN {X 0,Y 312.595,Z 361.16,A -85,B 0,C 180,E1 -15685.934,E2 -15685.934} C_VEL
LIN {X 0,Y 312.544,Z 361.175,A -85,B 0,C 180,E1 -15689.651,E2 -15689.651} C_VEL
LIN {X 0,Y 312.518,Z 361.174,A -85,B 0,C 180,E1 -15693.69,E2 -15693.69} C_VEL
